// TIA Portal project "Marmita CAPIC" (V14)

(* hardware
DEVICE "S7-1200 station_1"  S7-1200 Station
   slot 0: "Rack_0"  S7-1200 Rack  Rack  V1.0
   slot 1: "Marmita CAPIC"  CPU 1214C DC/DC/DC  6ES7 214-1AG40-0XB0  V4.2
   slot 2: "DI 16/DQ 16x24VDC_1"  6ES7 223-1BL32-0XB0  V2.0
   slot 3: "DI 16/DQ 16x24VDC_2"  6ES7 223-1BL32-0XB0  V2.0
   slot 4: "AI 8xRTD_1"  SM 1231 AI8 x RTD  6ES7 231-5PF32-0XB0  V2.0
   slot 5: "AI 4x13BIT_1"  6ES7 231-4HD32-0XB0  V2.0
   slot 6: "AQ 4x14BIT_1"  6ES7 232-4HD32-0XB0  V2.0
DEVICE "CSM"  SCALANCE X-Station
   slot 0: "Bastidor SCALANCE X"  Rail
   slot 0: "Switch_MARMITA"  6GK7 277-1AA10-0AA0
DEVICE "CSM_1"  SCALANCE X-Station
   slot 0: "Bastidor SCALANCE X"  Rail
   slot 0: "Switch_REFRIGERACION"  6GK7 277-1AA10-0AA0
DEVICE "HMI MARMITA CAPIC"  Dummy PC
   slot 1: "Interfaz PROFINET"  PN-IO
*)

// ===== PLC "Marmita CAPIC"  CPU 1214C DC/DC/DC =====

VAR_GLOBAL   // PLC tag table "Tabla de variables estándar"
   "Clock_Byte" AT %MB4000 : Byte;
   "Clock_10Hz" AT %M4000.0 : Bool;
   "Clock_5Hz" AT %M4000.1 : Bool;
   "Clock_2.5Hz" AT %M4000.2 : Bool;
   "Clock_2Hz" AT %M4000.3 : Bool;
   "Clock_1.25Hz" AT %M4000.4 : Bool;
   "Clock_1Hz" AT %M4000.5 : Bool;
   "Clock_0.625Hz" AT %M4000.6 : Bool;
   "Clock_0.5Hz" AT %M4000.7 : Bool;
   "System_Byte" AT %MB4001 : Byte;
   "FirstScan" AT %M4001.0 : Bool;
   "DiagStatusUpdate" AT %M4001.1 : Bool;
   "AlwaysTRUE" AT %M4001.2 : Bool;
   "AlwaysFALSE" AT %M4001.3 : Bool;
   "Flanc_Trig_P (1Hz)" AT %M0.1 : Bool;
   "m_Zumbador" AT %M0.2 : Bool;
END_VAR

VAR_GLOBAL   // PLC tag table "Entrades Digitals"
   "Elevador abaix" AT %I8.0 : Bool;
   "Elevador adalt" AT %I8.1 : Bool;
   "Marmita volcada" AT %I8.2 : Bool;
   "Marmita desvolcada" AT %I8.3 : Bool;
   "Tapa oberta" AT %I8.4 : Bool;
   "Tapa tancada" AT %I8.5 : Bool;
   "Sensor posicio pales" AT %I8.6 : Bool;
   "Modul XPS-DMB Elevador OK" AT %I0.0 : Bool;
   "Modul XPS-DMB Tapa OK" AT %I0.1 : Bool;
   "Modul XPS-AF P.E OK" AT %I0.2 : Bool;
   "Fallo Murr" AT %I0.3 : Bool;
   "Termistor motor pales" AT %I0.4 : Bool;
   "Termistor motor volcador" AT %I0.5 : Bool;
   "Fallo Magnetotermic variador pales" AT %I0.6 : Bool;
   "Fallo Magnetotermic variador volcador" AT %I0.7 : Bool;
   "Fallo Variador pales" AT %I1.0 : Bool;
   "Fallo Variador volcador" AT %I1.1 : Bool;
   "MARXA PROCES" AT %I10.0 : Bool;
   "PARADA PROCES" AT %I10.1 : Bool;
   "PAUSA PROCES" AT %I10.2 : Bool;
   "CT100 Contador Entrada Aigua Osmotitzada" AT %I1.5 : Bool;   // 1 impuls = 1 L
   "Boto Pujar Elevador" AT %I10.3 : Bool;
   "Boto Paro Elevador" AT %I10.4 : Bool;
   "Boto Baixar Elevador" AT %I10.5 : Bool;
   "Boto volcar marmita" AT %I10.6 : Bool;
   "Boto desvolcar marmita" AT %I10.7 : Bool;
   "Boto pujar tapa" AT %I11.0 : Bool;
   "Boto baixar tapa" AT %I11.1 : Bool;
   "Boto marxa pales" AT %I11.2 : Bool;
   "Boto paro pales" AT %I11.3 : Bool;
   "Boto marxa turmix" AT %I11.4 : Bool;
   "Boto paro turmix" AT %I11.5 : Bool;
   "Fallo Termic Elevador" AT %I1.2 : Bool;
END_VAR

VAR_GLOBAL   // PLC tag table "Sortides Digitals"
   "Color Verd" AT %Q0.0 : Bool;
   "Color Taronja" AT %Q0.1 : Bool;
   "Color Vermell" AT %Q0.2 : Bool;
   "Zumbador" AT %Q0.3 : Bool;
   "Pujar Elevador" AT %Q8.0 : Bool;
   "Baixar Elevador" AT %Q8.1 : Bool;
   "Volcar Marmita" AT %Q8.2 : Bool;
   "Desvolcar Marmita" AT %Q8.3 : Bool;
   "Pujar Tapa" AT %Q8.4 : Bool;
   "Baixar Tapa" AT %Q8.5 : Bool;
   "Motor Pales" AT %Q8.6 : Bool;
   "Motor Turmix" AT %Q8.7 : Bool;
   "EV Aire Comprimit" AT %Q9.0 : Bool;
   "EV107 Purga Camisa" AT %Q9.2 : Bool;
   "EV108 Aigua Osmotitzada" AT %Q9.1 : Bool;
   "EV101 Retorn Condensats Vapor" AT %Q9.3 : Bool;
   "EV102 Entrada Aero" AT %Q9.4 : Bool;
   "EV103 Retorn Aero" AT %Q9.5 : Bool;
   "EV104 Entrada Aigua Freda" AT %Q9.6 : Bool;
   "EV105 Retorn Aigua Freda" AT %Q9.7 : Bool;
END_VAR

VAR_GLOBAL   // PLC tag table "Entrades Analogiques"
   "BT100 Sonda Tº Entrada Vapor" AT %IW162 : Int;
   "BT101 Sonda Tº Condensats Vapor" AT %IW164 : Int;
   "BT102 Sonda Tº Entrada Aero" AT %IW166 : Int;
   "BT103 Sonda Tº Retorn Aero" AT %IW168 : Int;
   "BT104 Sonda Tº Entrada Aigua Freda" AT %IW170 : Int;
   "BT105 Sonda Tº Retorn Aigua Freda" AT %IW172 : Int;
   "BP100 Presostat Entrada Vapor" AT %IW112 : Int;
   "BP101 Presostat Condensats Vapor" AT %IW114 : Int;
   "BP102 Presostat Aire" AT %IW116 : Int;
   "Sonda Temperatura Producte" AT %IW160 : Int;
END_VAR

VAR_GLOBAL   // PLC tag table "Sortides Analogiques"
   "EV100 Entrada Vapor" AT %QW176 : Int;
END_VAR

VAR_GLOBAL   // PLC tag table "PID Vapor"
   "Distrurbance" AT %MD106 : Real;
   "ManualValve" AT %MD110 : Real;
   "ErrorAck" AT %M100.0 : Bool;
   "Input_PER" AT %MW102 : Int;
   "Setpoint" AT %MD114 : Real;
   "Input" AT %MD118 : Real;
   "ManualEnable" AT %M100.1 : Bool;
   "Error" AT %M100.2 : Bool;
   "Output_PER" AT %MW104 : Int;
END_VAR

TYPE "Plantilla Variables Receptes"
   STRUCT
      Nº_Recepta : USInt;
      "Consigna Temps Inicialtizacio Hores" : USInt;
      "Consigna Temps Inicialtizacio Minuts" : USInt;
      "Consigna Temperatura" : USInt;
      "Consigna Temperatura Refredament" : USInt;
   END_STRUCT;
END_TYPE

DATA_BLOCK "DB_Recetas"   // DB2
{ S7_Optimized_Access := 'FALSE' }
VERSION : 0.1
   VAR
      "Recepta Actual" : "Plantilla Variables Receptes";
      "Recepta 1" : "Plantilla Variables Receptes";
      "Recepta 2" : "Plantilla Variables Receptes";
      "Recepta 3" : "Plantilla Variables Receptes";
      "Recepta 4" : "Plantilla Variables Receptes";
      "Recepta 5" : "Plantilla Variables Receptes";
      "Recepta 6" : "Plantilla Variables Receptes";
      "Recepta 7" : "Plantilla Variables Receptes";
      "Recepta 8" : "Plantilla Variables Receptes";
      "Recepta 9" : "Plantilla Variables Receptes";
      "Recepta 10" : "Plantilla Variables Receptes";
      "Recepta 11" : "Plantilla Variables Receptes";
      "Recepta 12" : "Plantilla Variables Receptes";
      "Recepta 13" : "Plantilla Variables Receptes";
      "Recepta 14" : "Plantilla Variables Receptes";
      "Recepta 15" : "Plantilla Variables Receptes";
      "Recepta 16" : "Plantilla Variables Receptes";
      "Recepta 17" : "Plantilla Variables Receptes";
      "Recepta 18" : "Plantilla Variables Receptes";
      "Recepta 19" : "Plantilla Variables Receptes";
      "Recepta 20" : "Plantilla Variables Receptes";
      "Recepta 21" : "Plantilla Variables Receptes";
      "Recepta 22" : "Plantilla Variables Receptes";
      "Recepta 23" : "Plantilla Variables Receptes";
      "Recepta 24" : "Plantilla Variables Receptes";
      "Recepta 25" : "Plantilla Variables Receptes";
      "Recepta 26" : "Plantilla Variables Receptes";
      "Recepta 27" : "Plantilla Variables Receptes";
      "Recepta 28" : "Plantilla Variables Receptes";
      "Recepta 29" : "Plantilla Variables Receptes";
      "Recepta 30" : "Plantilla Variables Receptes";
   END_VAR
BEGIN
END_DATA_BLOCK

DATA_BLOCK "Contador hores funcionament pales"   // DB3
{ S7_Optimized_Access := 'TRUE' }
VERSION : 0.1
// stored: InstanceOfName Contador hores de funcionament
"Contador hores de funcionament"
BEGIN
END_DATA_BLOCK

DATA_BLOCK "FB Pales_DB"   // DB4
{ S7_Optimized_Access := 'TRUE' }
VERSION : 0.1
// stored: InstanceOfName FB Pales
"FB Pales"
BEGIN
END_DATA_BLOCK

DATA_BLOCK "Control Coccio_DB"   // DB5
{ S7_Optimized_Access := 'TRUE' }
VERSION : 0.1
// stored: InstanceOfName Control Coccio
"Control Coccio"
BEGIN
END_DATA_BLOCK

DATA_BLOCK "Asignar Receptes_DB"   // DB6
{ S7_Optimized_Access := 'FALSE' }
VERSION : 0.1
// stored: InstanceOfName Asignar Receptes
"Asignar Receptes"
BEGIN
END_DATA_BLOCK

DATA_BLOCK "Intermitencia Ajustable_Zumbador_Fase_1"   // DB7
{ S7_Optimized_Access := 'TRUE' }
VERSION : 0.1
// stored: InstanceOfName Intermitencia Ajustable
"Intermitencia Ajustable"
BEGIN
END_DATA_BLOCK

DATA_BLOCK "DB_Variables_Estats"   // DB11
{ S7_Optimized_Access := 'FALSE' }
VERSION : 0.1
   VAR
      Control_Coccio : Struct
         "Estat Proces" : Bool;
         "Status Proces" : String;
      END_STRUCT;
   END_VAR
BEGIN
END_DATA_BLOCK

DATA_BLOCK "Contador aigua osmotitzada_DB"   // DB13
{ S7_Optimized_Access := 'TRUE' }
VERSION : 0.1
// stored: InstanceOfName Contador aigua osmotitzada
"Contador aigua osmotitzada"
BEGIN
END_DATA_BLOCK

DATA_BLOCK "DB_Varaibles_Pantalla"   // DB14
{ S7_Optimized_Access := 'FALSE' }
VERSION : 0.1
   VAR
      "Botons Generals" : Struct
         "Cargar Receta" : Bool;   // Carrega la recepta
      END_STRUCT;
      "Contador aigua osmotitzada" : Struct
         "Marxa Entrada Aigua" : Bool;   // Aigua osmotitzada
         "Paro Entrada Aigua" : Bool;   // Aigua osmotitzada
         "Reset Contador" : Bool;
         "Consigna Litros para Entrar" : SInt;
         "Valor contador" : SInt;
      END_STRUCT;
      "Ajustes Cocció" : Struct
         "Temps de Neteja" : SInt := 120;   // Temps de proces de neteja (segons)
      END_STRUCT;
      "Botons Manual" : Struct
         "Modo Manual" : Bool;
         "Pujar Elevador" : Bool;
         "Baixar Elevador" : Bool;
         "Volcar marmita" : Bool;
         "Desvolcar marmita" : Bool;
         "Pujar tapa" : Bool;
         "Baixar tapa" : Bool;
         "Pales ON/OFF" : Bool;
         "Tuemix ON/OFF" : Bool;
         "EV Aire" : Bool;
         "EV Aigua Freda" : Bool;
         "EV Aero" : Bool;
         "EV Purga" : Bool;
         "EV Aigua osmotitzada" : Bool;
      END_STRUCT;
   END_VAR
BEGIN
END_DATA_BLOCK

// folder: System blocks/Program resources

DATA_BLOCK "Timer_1"   // DB8
{ S7_Optimized_Access := 'TRUE' }
AUTHOR : Simatic
FAMILY : IEC
NAME : IEC_TMR
VERSION : 1.0
// stored: InstanceOfName IEC_TIMER
"IEC_TIMER"
BEGIN
END_DATA_BLOCK

DATA_BLOCK "Timer_2"   // DB9
{ S7_Optimized_Access := 'TRUE' }
AUTHOR : Simatic
FAMILY : IEC
NAME : IEC_TMR
VERSION : 1.0
// stored: InstanceOfName IEC_TIMER
"IEC_TIMER"
BEGIN
END_DATA_BLOCK

DATA_BLOCK "TM_Impuls"   // DB17
{ S7_Optimized_Access := 'TRUE' }
AUTHOR : Simatic
FAMILY : IEC
NAME : IEC_TMR
VERSION : 1.0
// stored: InstanceOfName IEC_TIMER
"IEC_TIMER"
BEGIN
END_DATA_BLOCK

// folder: (top level)

FUNCTION_BLOCK "Contador hores de funcionament"   // FB1, LAD
{ S7_Optimized_Access := 'TRUE' }
VERSION : 0.1
   VAR_INPUT
      "Entrada cicle 1 Hz" : Bool;
      "Variable de vigilancia" : Bool;
      "Valor de avis" : Time;
      "Reset Contador" : Bool;
   END_VAR
   VAR_OUTPUT
      "t Acumulat TIME" : Time;
      "t Acumulat DINT (ms)" : DInt;
      "t Manteniment TIME" : Time;
      "t Manteniment DINT (ms)" : DInt;
      "Avis de Manteniment" : Bool;
   END_VAR
   VAR
      Trig_Contador : Bool;
   END_VAR
   VAR RETAIN
      Val_Cont_Acumulat : DInt;
      Val_Cont_Manteniment : DInt;
   END_VAR
   VAR_TEMP
      temp : DInt;
   END_VAR
   VAR_TEMP   // added for the SCL form of the ladder/FBD networks
      _w1 : Bool;
      _w2 : Bool;
   END_VAR
BEGIN

REGION Network 1: Contador Acumulat
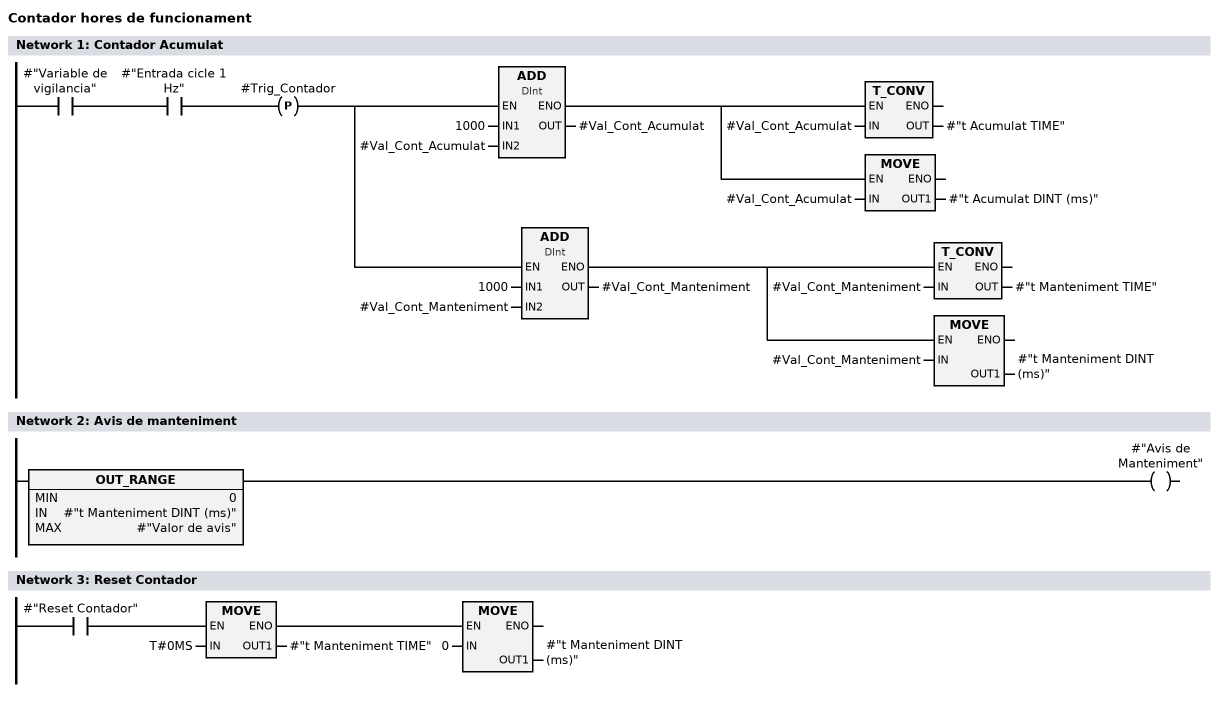
   #_w1 := #"Variable de vigilancia" AND #"Entrada cicle 1 Hz";
   #_w2 := #_w1 AND NOT #Trig_Contador;   // rising edge
   #Trig_Contador := #_w1;
   IF #_w2 THEN
       #Val_Cont_Acumulat := 1000 + #Val_Cont_Acumulat;
       #"t Acumulat TIME" := T_CONV(IN := #Val_Cont_Acumulat);
       #"t Acumulat DINT (ms)" := #Val_Cont_Acumulat;
       #Val_Cont_Manteniment := 1000 + #Val_Cont_Manteniment;
       #"t Manteniment TIME" := T_CONV(IN := #Val_Cont_Manteniment);
       #"t Manteniment DINT (ms)" := #Val_Cont_Manteniment;
   END_IF;
END_REGION

REGION Network 2: Avis de manteniment
   #"Avis de Manteniment" := (#"t Manteniment DINT (ms)" < 0) OR (#"t Manteniment DINT (ms)" > #"Valor de avis");
END_REGION

REGION Network 3: Reset Contador
   RUNG wire#powerrail
      Contact( #"Reset Contador" )
      Move(in := T#0MS, out1 => #"t Manteniment TIME")
      Move(in := 0, out1 => #"t Manteniment DINT (ms)")
   END_RUNG
   // the same network as SCL:
   IF #"Reset Contador" THEN
       #"t Manteniment TIME" := T#0MS;
       #"t Manteniment DINT (ms)" := 0;
   END_IF;
END_REGION
END_FUNCTION_BLOCK

FUNCTION_BLOCK "FB_Neteja_Camisa"   // FB2, LAD
{ S7_Optimized_Access := 'TRUE' }
VERSION : 0.1
   VAR_INPUT
      Start : Bool;
      Pausa : Bool;
      "Condicio Marxa" : Bool;
      "Clock 1 hz" : Bool;
      "Consigna Temps Neteja" : Time := T#0MS;
   END_VAR
   VAR_OUTPUT
      "EV Aire Comprimit" : Bool;
      "EV Purga" : Bool;
      Status : String;
      "Proces ON/OFF" : Bool;
      "Fin Proces" : Bool;
   END_VAR
   VAR RETAIN
      Contador_Temps_Acum : DInt;
   END_VAR
   VAR
      Trig_Start : Bool;
      Trig_1s : Bool;
      Trig_Fin : Bool;
   END_VAR
   VAR RETAIN
      En_Pausa : Bool;
      "Proces Neteja" : Bool;
   END_VAR
   VAR_TEMP
      Temp_BOOL : Bool;
      Temp_INT : Int;
      Temp_REAL : Real;
      Temp_DINT : DInt;
   END_VAR
   VAR_TEMP   // added for the SCL form of the ladder/FBD networks
      _w1 : Bool;
      _w2 : Bool;
   END_VAR
BEGIN

REGION Network 1: Inici Proces
   // Reset de Contador_Temps_Acum
   // Si condicio esta be, arranquem el proces
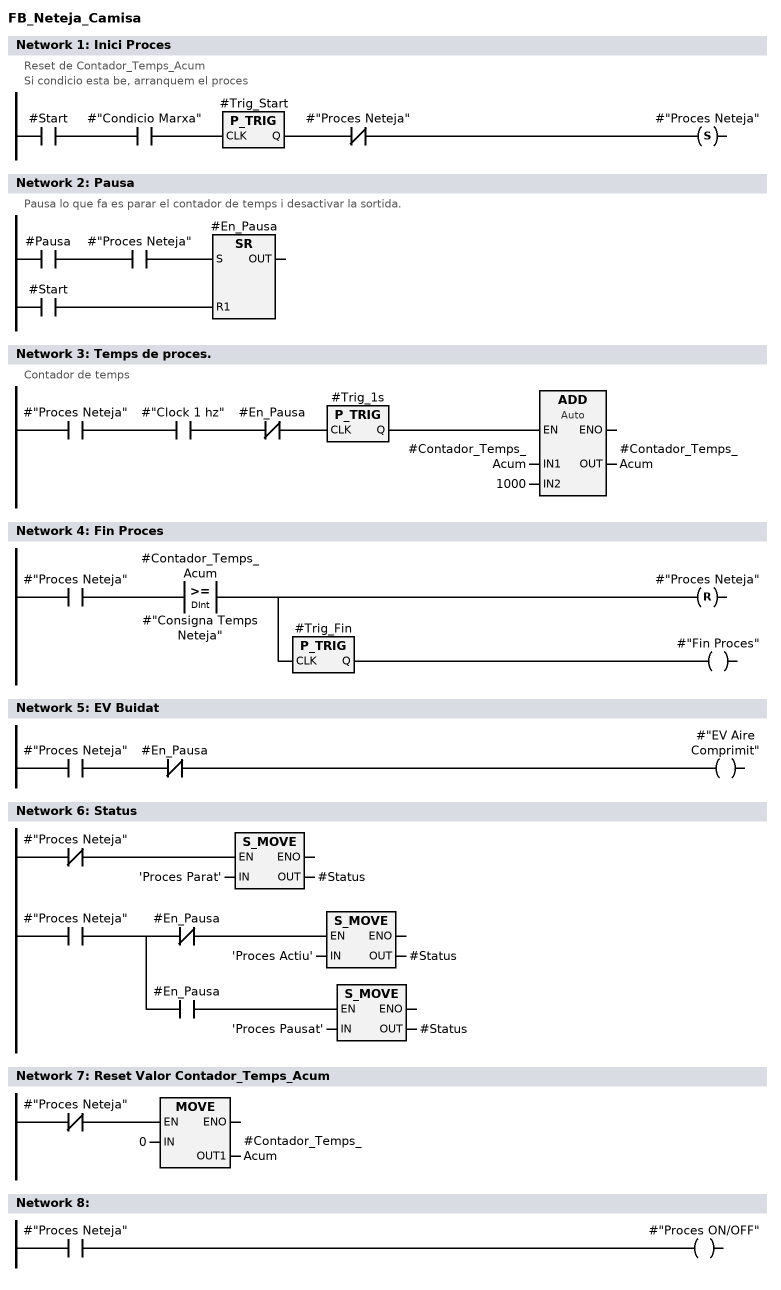
   RUNG wire#powerrail
      Contact( #Start )
      Contact( #"Condicio Marxa" )
      P_Trig( #Trig_Start )
      I_Contact( #"Proces Neteja" )
      S_Coil( #"Proces Neteja" )
   END_RUNG
   // the same network as SCL:
   #_w1 := #Start AND #"Condicio Marxa";
   #_w2 := #_w1 AND NOT #Trig_Start;   // rising edge
   #Trig_Start := #_w1;
   IF #_w2 AND NOT #"Proces Neteja" THEN #"Proces Neteja" := TRUE; END_IF;
END_REGION

REGION Network 2: Pausa
   // Pausa lo que fa es parar el contador de temps i desactivar la sortida.
   RUNG wire#powerrail
      Contact( #Pausa )
      Contact( #"Proces Neteja" )
      S_SR(operand := #En_Pausa, r1 := wire#w1)
   END_RUNG
   RUNG wire#powerrail
      Contact( #Start )
   END_RUNG wire#w1
   // the same network as SCL:
   IF #Pausa AND #"Proces Neteja" THEN
       #En_Pausa := TRUE;   // SR flip-flop
   END_IF;
   IF #Start THEN #En_Pausa := FALSE; END_IF;
END_REGION

REGION Network 3: Temps de proces.
   // Contador de temps
   RUNG wire#powerrail
      Contact( #"Proces Neteja" )
      Contact( #"Clock 1 hz" )
      I_Contact( #En_Pausa )
      P_Trig( #Trig_1s )
      Add(in1 := #Contador_Temps_Acum, in2 := 1000, out => #Contador_Temps_Acum)
   END_RUNG
   // the same network as SCL:
   #_w1 := #"Proces Neteja" AND #"Clock 1 hz" AND NOT #En_Pausa;
   #_w2 := #_w1 AND NOT #Trig_1s;   // rising edge
   #Trig_1s := #_w1;
   IF #_w2 THEN #Contador_Temps_Acum := #Contador_Temps_Acum + 1000; END_IF;
END_REGION

REGION Network 4: Fin Proces
   RUNG wire#powerrail
      Contact( #"Proces Neteja" )
      { S7_Templates := "SrcType := DInt" } GE_Contact(in1 := #Contador_Temps_Acum, in2 := #"Consigna Temps Neteja")
      wire#w1
      R_Coil( #"Proces Neteja" )
   END_RUNG
   RUNG wire#w1
      P_Trig( #Trig_Fin )
      Coil( #"Fin Proces" )
   END_RUNG
   // the same network as SCL:
   #_w1 := #"Proces Neteja" AND (#Contador_Temps_Acum >= #"Consigna Temps Neteja");
   IF #_w1 THEN #"Proces Neteja" := FALSE; END_IF;
   #_w2 := #_w1 AND NOT #Trig_Fin;   // rising edge
   #Trig_Fin := #_w1;
   #"Fin Proces" := #_w2;
END_REGION

REGION Network 5: EV Buidat
   RUNG wire#powerrail
      Contact( #"Proces Neteja" )
      I_Contact( #En_Pausa )
      Coil( #"EV Aire Comprimit" )
   END_RUNG
   // the same network as SCL:
   #"EV Aire Comprimit" := #"Proces Neteja" AND NOT #En_Pausa;
END_REGION

REGION Network 6: Status
   IF NOT #"Proces Neteja" THEN S_MOVE(in := 'Proces Parat', out => #Status); END_IF;
   IF #"Proces Neteja" AND NOT #En_Pausa THEN S_MOVE(in := 'Proces Actiu', out => #Status); END_IF;
   IF #"Proces Neteja" AND #En_Pausa THEN S_MOVE(in := 'Proces Pausat', out => #Status); END_IF;
END_REGION

REGION Network 7: Reset Valor Contador_Temps_Acum
   RUNG wire#powerrail
      I_Contact( #"Proces Neteja" )
      Move(in := 0, out1 => #Contador_Temps_Acum)
   END_RUNG
   // the same network as SCL:
   IF NOT #"Proces Neteja" THEN #Contador_Temps_Acum := 0; END_IF;
END_REGION

REGION Network 8
   RUNG wire#powerrail
      Contact( #"Proces Neteja" )
      Coil( #"Proces ON/OFF" )
   END_RUNG
   // the same network as SCL:
   #"Proces ON/OFF" := #"Proces Neteja";
END_REGION
END_FUNCTION_BLOCK

FUNCTION_BLOCK "FB Pales"   // FB4, LAD
{ S7_Optimized_Access := 'TRUE' }
VERSION : 0.1
   VAR_INPUT
      Marxa : Bool;
      Paro : Bool;
      "Condicio Marxa" : Bool;
      "Fallo Termic" : Bool;
      "Fallo Variador" : Bool;
      "Ref. Velocitat" : Int;
   END_VAR
   VAR_OUTPUT
      "Marxa Variador" : Bool;
      "OUT: Velocitat" : Int;
      "Proces ON/OFF" : Bool;
      Status : String;
   END_VAR
   VAR RETAIN
      Contador_Temps_Acum : DInt;
   END_VAR
   VAR
      Trig_Start : Bool;
      Trig_1s : Bool;
      Trig_Fin : Bool;
      "Motor Pales" : Bool;
   END_VAR
   VAR_TEMP
      Temp_Int : Int;
      Temp_Dint : DInt;
      Temp_Real : Real;
      Temp_Bool : Bool;
   END_VAR
   VAR_TEMP   // added for the SCL form of the ladder/FBD networks
      _w1 : Bool;
      _w2 : Bool;
   END_VAR
BEGIN

REGION Network 1: Inici Proces
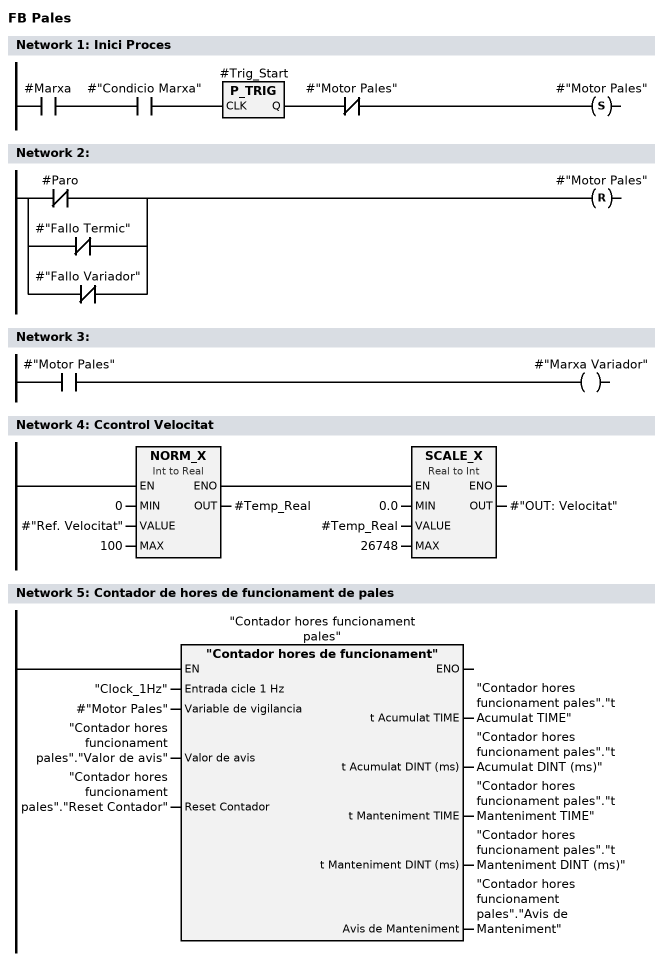
   RUNG wire#powerrail
      Contact( #Marxa )
      Contact( #"Condicio Marxa" )
      P_Trig( #Trig_Start )
      I_Contact( #"Motor Pales" )
      S_Coil( #"Motor Pales" )
   END_RUNG
   // the same network as SCL:
   #_w1 := #Marxa AND #"Condicio Marxa";
   #_w2 := #_w1 AND NOT #Trig_Start;   // rising edge
   #Trig_Start := #_w1;
   IF #_w2 AND NOT #"Motor Pales" THEN #"Motor Pales" := TRUE; END_IF;
END_REGION

REGION Network 2
   RUNG wire#powerrail
      I_Contact( #Paro )
      wire#w1
      R_Coil( #"Motor Pales" )
   END_RUNG
   RUNG wire#powerrail
      I_Contact( #"Fallo Termic" )
   END_RUNG wire#w1
   RUNG wire#powerrail
      I_Contact( #"Fallo Variador" )
   END_RUNG wire#w1
   // the same network as SCL:
   IF NOT #Paro OR NOT #"Fallo Termic" OR NOT #"Fallo Variador" THEN #"Motor Pales" := FALSE; END_IF;
END_REGION

REGION Network 3
   RUNG wire#powerrail
      Contact( #"Motor Pales" )
      Coil( #"Marxa Variador" )
   END_RUNG
   // the same network as SCL:
   #"Marxa Variador" := #"Motor Pales";
END_REGION

REGION Network 4: Ccontrol Velocitat
   RUNG wire#powerrail
      { S7_Templates := "[SrcType := Int, DestType := Real]" } Normalize(min := 0, value := #"Ref. Velocitat", max := 100, out => #Temp_Real)
      { S7_Templates := "[SrcType := Real, DestType := Int]" } Scale(min := 0.0, value := #Temp_Real, max := 26748, out => #"OUT: Velocitat")
   END_RUNG
   // the same network as SCL:
   #Temp_Real := NORM_X(MIN := 0, VALUE := #"Ref. Velocitat", MAX := 100);
   #"OUT: Velocitat" := SCALE_X(MIN := 0.0, VALUE := #Temp_Real, MAX := 26748);
END_REGION

REGION Network 5: Contador de hores de funcionament de pales
   RUNG wire#powerrail
      "Contador hores funcionament pales"("Entrada cicle 1 Hz" := "Clock_1Hz", "Variable de vigilancia" := #"Motor Pales", "Valor de avis" := "Contador hores funcionament pales"."Valor de avis", "Reset Contador" := "Contador hores funcionament pales"."Reset Contador", "t Acumulat TIME" => "Contador hores funcionament pales"."t Acumulat TIME", "t Acumulat DINT (ms)" => "Contador hores funcionament pales"."t Acumulat DINT (ms)", "t Manteniment TIME" => "Contador hores funcionament pales"."t Manteniment TIME", "t Manteniment DINT (ms)" => "Contador hores funcionament pales"."t Manteniment DINT (ms)", "Avis de Manteniment" => "Contador hores funcionament pales"."Avis de Manteniment")
   END_RUNG
   // the same network as SCL:
   "Contador hores funcionament pales"("Entrada cicle 1 Hz" := "Clock_1Hz",   // "Contador hores de funcionament"
                           "Variable de vigilancia" := #"Motor Pales",
                           "Valor de avis" := "Contador hores funcionament pales"."Valor de avis",
                           "Reset Contador" := "Contador hores funcionament pales"."Reset Contador",
                           "t Acumulat TIME" => "Contador hores funcionament pales"."t Acumulat TIME",
                           "t Acumulat DINT (ms)" => "Contador hores funcionament pales"."t Acumulat DINT (ms)",
                           "t Manteniment TIME" => "Contador hores funcionament pales"."t Manteniment TIME",
                           "t Manteniment DINT (ms)" => "Contador hores funcionament pales"."t Manteniment DINT (ms)",
                           "Avis de Manteniment" => "Contador hores funcionament pales"."Avis de Manteniment");
END_REGION
END_FUNCTION_BLOCK

FUNCTION_BLOCK "Control Coccio"   // FB8, LAD
{ S7_Optimized_Access := 'TRUE' }
VERSION : 0.1
   VAR_INPUT
      START : Bool;
      STOP : Bool;
      PAUSA : Bool;
      "Silenciar Alarma" : Bool;
      "Condicio Marxa Fase 1" : Bool;
      "Condicio Marxa Fase 2" : Bool;
      "Condicio Marxa Fase 3" : Bool;
      "Condicio Marxa Fase 4" : Bool;
      "Condicio Marxa Fase 5" : Bool;
      "Condicio Marxa Fase 6" : Bool;
      "Sonda Temperatura Producte" : USInt := 0;
      "Clock 1Hz" : Bool;
      "Receta Actual" : "Plantilla Variables Receptes";
      "Consigna Temps Neteja" : UDInt := 120;
   END_VAR
   VAR_OUTPUT
      "Estat Proces" : Bool;
      "Status Proces" : String;
   END_VAR
   VAR_IN_OUT
      Zumbador : Bool;
   END_VAR
   VAR
      M_Zumbador_Fase_1 : Bool;   // Zumbador de Avis de fin de fases i fin de procesos.
      M_Zumbador_Fase_2 : Bool;
      M_Zumbador_Fase_3 : Bool;
      M_Zumbador_Fase_4 : Bool;
      M_Zumbador_Fase_5 : Bool;
      M_Zumbador_Fase_6 : Bool;
      M_Zumbador_Fase_7 : Bool;
      M_Zumbador_Fase_8 : Bool;
      M_Zumbador_Fase_9 : Bool;
      M_Zumbador_Fase_10 : Bool;
   END_VAR
   VAR RETAIN
      M_Start : Bool;
      M_Pausa : Bool;
      "Nº Proces Actual" : USInt := 0;
      "Contador Fase 1" : UDInt;
      "Contador Fase 2" : UDInt;
      "Contador Fase 3" : UDInt;
      "Contador Fase 4" : UDInt;
      "Contador Fase 5" : UDInt;
      "Contador Fase 6" : UDInt;
      "Contador Fase 7" : UDInt;
      "Contador Fase 8" : UDInt;
      "Contador Fase 9" : UDInt;
      "Contador Fase 10" : UDInt;
      SR_Fase_1 : Bool;
      SR_Fase_2 : Bool;
      SR_Fase_3 : Bool;
      SR_Fase_4 : Bool;
      SR_Fase_5 : Bool;
      SR_Fase_6 : Bool;
      SR_Fase_7 : Bool;
      SR_Fase_8 : Bool;
      SR_Fase_9 : Bool;
      SR_Fase_10 : Bool;
   END_VAR
   VAR
      Flanc_inici_programa : Bool;
      Flanc_pausa_OFF : Bool;
      Flanc_Add_Fase_1 : Bool;
      Flanc_Add_Fase_2 : Bool;
      Flanc_Add_Fase_3 : Bool;
      Flanc_Add_Fase_4 : Bool;
      Flanc_Add_Fase_5 : Bool;
      Flanc_Add_Fase_6 : Bool;
      Flanc_Add_Fase_7 : Bool;
      Flanc_Add_Fase_8 : Bool;
      Flanc_Add_Fase_9 : Bool;
      Flanc_Add_Fase_10 : Bool;
      Buffer_Sonda_Temperatura_Producte : USInt;
      Intermitencia : Bool;
      Temp_MAX : USInt;
      "Temperatura Estable" : Bool;
   END_VAR
   VAR RETAIN
      "Conv Temps a segons" : UDInt;
   END_VAR
   VAR_TEMP
      Temp_TIME : Time;
      Temp_USINT : USInt;
   END_VAR
   VAR_TEMP   // added for the SCL form of the ladder/FBD networks
      _w1 : Bool;
      _w2 : Bool;
      _w3 : Bool;
      _w4 : Bool;
   END_VAR
BEGIN

REGION Network 1: Marxa sequencia.
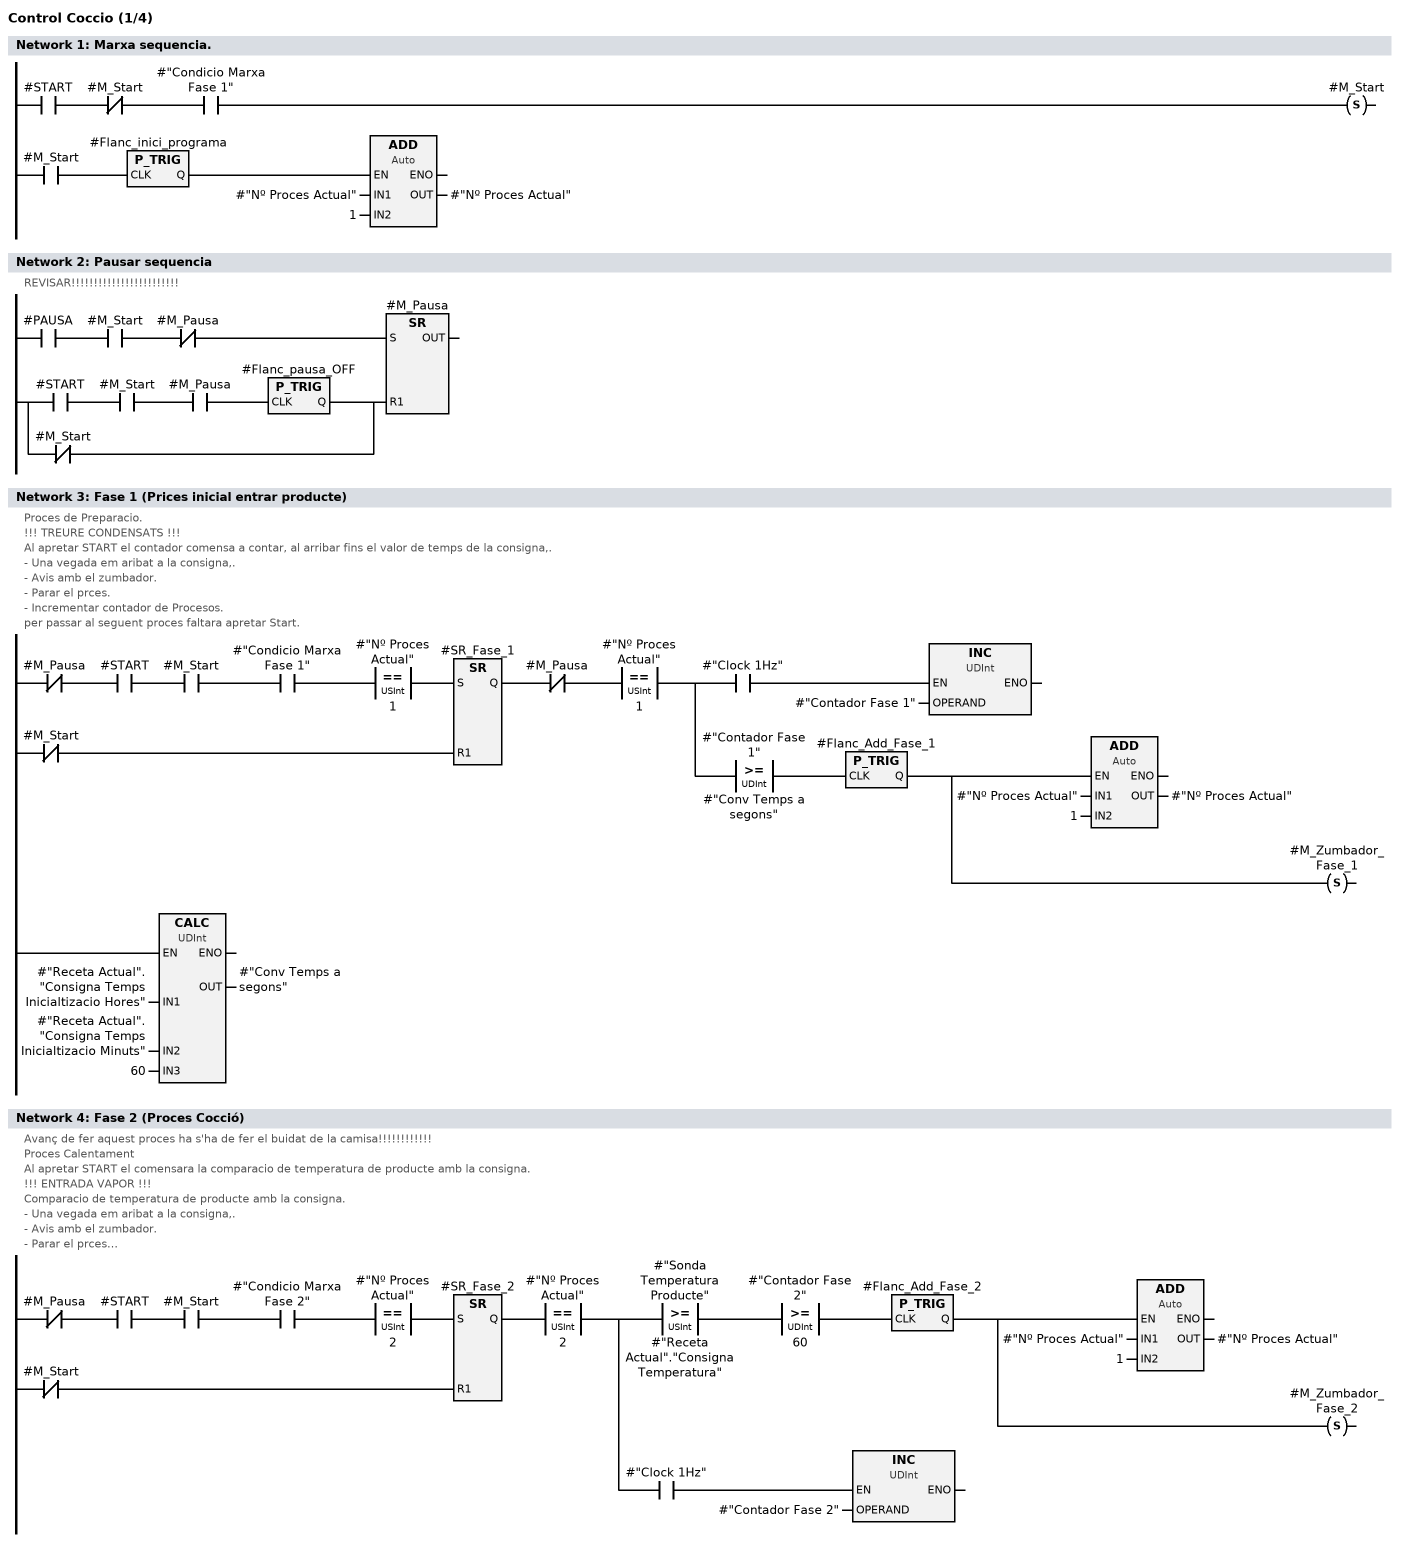
   RUNG wire#powerrail
      Contact( #START )
      I_Contact( #M_Start )
      Contact( #"Condicio Marxa Fase 1" )
      S_Coil( #M_Start )
   END_RUNG
   RUNG wire#powerrail
      Contact( #M_Start )
      P_Trig( #Flanc_inici_programa )
      Add(in1 := #"Nº Proces Actual", in2 := 1, out => #"Nº Proces Actual")
   END_RUNG
   // the same network as SCL:
   IF #START AND NOT #M_Start AND #"Condicio Marxa Fase 1" THEN #M_Start := TRUE; END_IF;
   #_w1 := #M_Start AND NOT #Flanc_inici_programa;   // rising edge
   #Flanc_inici_programa := #M_Start;
   IF #_w1 THEN #"Nº Proces Actual" := #"Nº Proces Actual" + 1; END_IF;
END_REGION

REGION Network 2: Pausar sequencia
   // REVISAR!!!!!!!!!!!!!!!!!!!!!!!!
   RUNG wire#powerrail
      Contact( #PAUSA )
      Contact( #M_Start )
      I_Contact( #M_Pausa )
      S_SR(operand := #M_Pausa, r1 := wire#w1)
   END_RUNG
   RUNG wire#powerrail
      Contact( #START )
      Contact( #M_Start )
      Contact( #M_Pausa )
      P_Trig( #Flanc_pausa_OFF )
   END_RUNG wire#w1
   RUNG wire#powerrail
      I_Contact( #M_Start )
   END_RUNG wire#w1
   // the same network as SCL:
   #_w1 := #START AND #M_Start AND #M_Pausa;
   #_w2 := #_w1 AND NOT #Flanc_pausa_OFF;   // rising edge
   #Flanc_pausa_OFF := #_w1;
   IF #PAUSA AND #M_Start AND NOT #M_Pausa THEN
       #M_Pausa := TRUE;   // SR flip-flop
   END_IF;
   IF #_w2 OR NOT #M_Start THEN #M_Pausa := FALSE; END_IF;
END_REGION

REGION Network 3: Fase 1 (Prices inicial entrar producte)
   // Proces de Preparacio.
   // 
   // !!! TREURE CONDENSATS !!!
   // 
   // Al apretar START el contador comensa a contar, al arribar fins el valor de temps de la consigna,.
   // 
   // - Una vegada em aribat a la consigna,.
   // - Avis amb el zumbador.
   // - Parar el prces.
   // - Incrementar contador de Procesos.
   // 
   // per passar al seguent proces faltara apretar Start.
   IF NOT #M_Pausa AND #START AND #M_Start AND #"Condicio Marxa Fase 1" AND (#"Nº Proces Actual" = 1) THEN
       #SR_Fase_1 := TRUE;   // SR flip-flop
   END_IF;
   IF NOT #M_Start THEN #SR_Fase_1 := FALSE; END_IF;
   #_w1 := #SR_Fase_1 AND NOT #M_Pausa AND (#"Nº Proces Actual" = 1);
   IF #_w1 AND #"Clock 1Hz" THEN #"Contador Fase 1" := #"Contador Fase 1" + 1; END_IF;
   #_w2 := #_w1 AND (#"Contador Fase 1" >= #"Conv Temps a segons");
   #_w3 := #_w2 AND NOT #Flanc_Add_Fase_1;   // rising edge
   #Flanc_Add_Fase_1 := #_w2;
   IF #_w3 THEN
       #"Nº Proces Actual" := #"Nº Proces Actual" + 1;
       #M_Zumbador_Fase_1 := TRUE;
   END_IF;
   CALC(in1 := #"Receta Actual"."Consigna Temps Inicialtizacio Hores",
        in2 := #"Receta Actual"."Consigna Temps Inicialtizacio Minuts",
        in3 := 60,
        out => #"Conv Temps a segons");
END_REGION

REGION Network 4: Fase 2 (Proces Cocció)
   // Avanç de fer aquest proces ha s'ha de fer el buidat de la camisa!!!!!!!!!!!!
   // 
   // Proces Calentament
   // 
   // Al apretar START el comensara la comparacio de temperatura de producte amb la consigna.
   // 
   // !!! ENTRADA VAPOR !!!
   // 
   // Comparacio de temperatura de producte amb la consigna.
   // 
   // - Una vegada em aribat a la consigna,.
   // - Avis amb el zumbador.
   // - Parar el prces.
   // - Incrementar contador de Procesos.
   RUNG wire#powerrail
      I_Contact( #M_Pausa )
      Contact( #START )
      Contact( #M_Start )
      Contact( #"Condicio Marxa Fase 2" )
      { S7_Templates := "SrcType := USInt" } EQ_Contact(in1 := #"Nº Proces Actual", in2 := 2)
      S_SR(operand := #SR_Fase_2, r1 := wire#w1)
      { S7_Templates := "SrcType := USInt" } EQ_Contact(in1 := #"Nº Proces Actual", in2 := 2)
      wire#w2
      { S7_Templates := "SrcType := USInt" } GE_Contact(in1 := #"Sonda Temperatura Producte", in2 := #"Receta Actual"."Consigna Temperatura")
      { S7_Templates := "SrcType := UDInt" } GE_Contact(in1 := #"Contador Fase 2", in2 := 60)
      P_Trig( #Flanc_Add_Fase_2 )
      wire#w3
      Add(in1 := #"Nº Proces Actual", in2 := 1, out => #"Nº Proces Actual")
   END_RUNG
   RUNG wire#powerrail
      I_Contact( #M_Start )
   END_RUNG wire#w1
   RUNG wire#w3
      S_Coil( #M_Zumbador_Fase_2 )
   END_RUNG
   RUNG wire#w2
      Contact( #"Clock 1Hz" )
      { S7_Templates := "DestType := UDInt" } Inc( #"Contador Fase 2" )
   END_RUNG
   // the same network as SCL:
   IF NOT #M_Pausa AND #START AND #M_Start AND #"Condicio Marxa Fase 2" AND (#"Nº Proces Actual" = 2) THEN
       #SR_Fase_2 := TRUE;   // SR flip-flop
   END_IF;
   IF NOT #M_Start THEN #SR_Fase_2 := FALSE; END_IF;
   #_w1 := #SR_Fase_2 AND (#"Nº Proces Actual" = 2);
   #_w2 := #_w1 AND (#"Sonda Temperatura Producte" >= #"Receta Actual"."Consigna Temperatura") AND (#"Contador Fase 2" >= 60);
   #_w3 := #_w2 AND NOT #Flanc_Add_Fase_2;   // rising edge
   #Flanc_Add_Fase_2 := #_w2;
   IF #_w3 THEN
       #"Nº Proces Actual" := #"Nº Proces Actual" + 1;
       #M_Zumbador_Fase_2 := TRUE;
   END_IF;
   IF #_w1 AND #"Clock 1Hz" THEN #"Contador Fase 2" := #"Contador Fase 2" + 1; END_IF;
END_REGION

REGION Network 5: Fase 3 (Neteja)
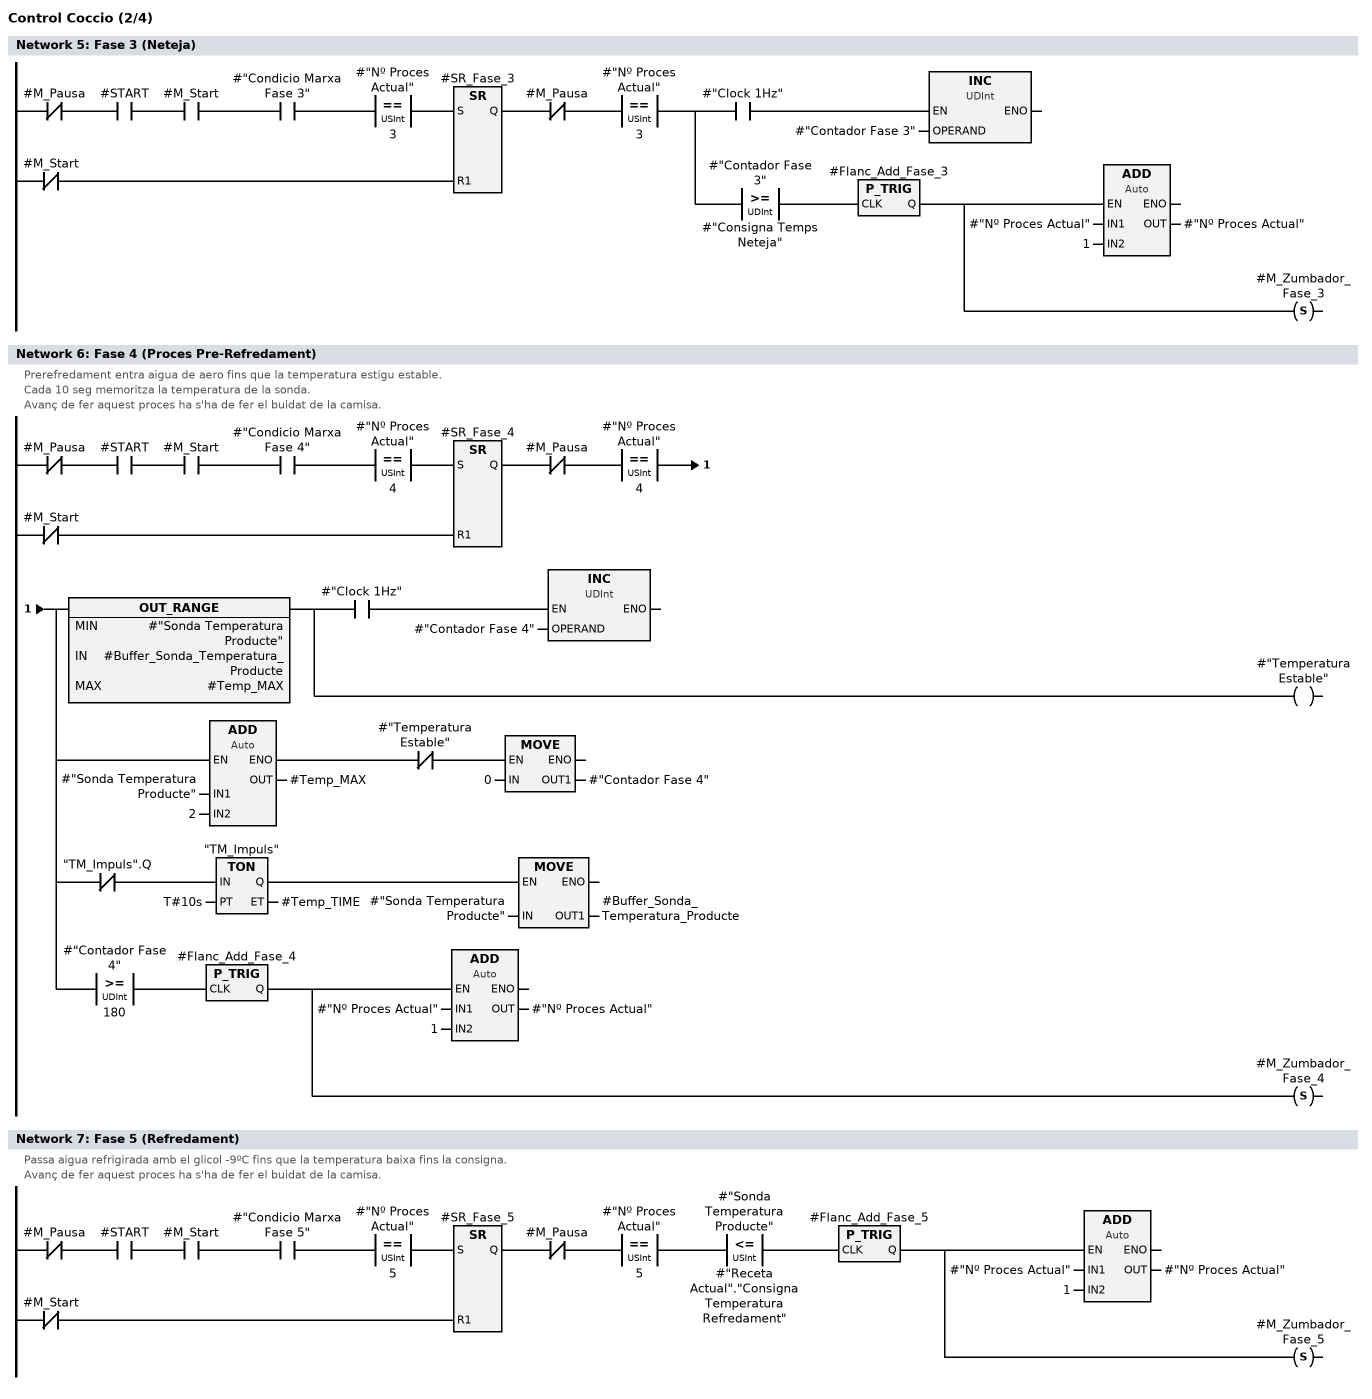
   RUNG wire#powerrail
      I_Contact( #M_Pausa )
      Contact( #START )
      Contact( #M_Start )
      Contact( #"Condicio Marxa Fase 3" )
      { S7_Templates := "SrcType := USInt" } EQ_Contact(in1 := #"Nº Proces Actual", in2 := 3)
      S_SR(operand := #SR_Fase_3, r1 := wire#w1)
      I_Contact( #M_Pausa )
      { S7_Templates := "SrcType := USInt" } EQ_Contact(in1 := #"Nº Proces Actual", in2 := 3)
      wire#w2
      Contact( #"Clock 1Hz" )
      { S7_Templates := "DestType := UDInt" } Inc( #"Contador Fase 3" )
   END_RUNG
   RUNG wire#powerrail
      I_Contact( #M_Start )
   END_RUNG wire#w1
   RUNG wire#w2
      { S7_Templates := "SrcType := UDInt" } GE_Contact(in1 := #"Contador Fase 3", in2 := #"Consigna Temps Neteja")
      P_Trig( #Flanc_Add_Fase_3 )
      wire#w3
      Add(in1 := #"Nº Proces Actual", in2 := 1, out => #"Nº Proces Actual")
   END_RUNG
   RUNG wire#w3
      S_Coil( #M_Zumbador_Fase_3 )
   END_RUNG
   // the same network as SCL:
   IF NOT #M_Pausa AND #START AND #M_Start AND #"Condicio Marxa Fase 3" AND (#"Nº Proces Actual" = 3) THEN
       #SR_Fase_3 := TRUE;   // SR flip-flop
   END_IF;
   IF NOT #M_Start THEN #SR_Fase_3 := FALSE; END_IF;
   #_w1 := #SR_Fase_3 AND NOT #M_Pausa AND (#"Nº Proces Actual" = 3);
   IF #_w1 AND #"Clock 1Hz" THEN #"Contador Fase 3" := #"Contador Fase 3" + 1; END_IF;
   #_w2 := #_w1 AND (#"Contador Fase 3" >= #"Consigna Temps Neteja");
   #_w3 := #_w2 AND NOT #Flanc_Add_Fase_3;   // rising edge
   #Flanc_Add_Fase_3 := #_w2;
   IF #_w3 THEN
       #"Nº Proces Actual" := #"Nº Proces Actual" + 1;
       #M_Zumbador_Fase_3 := TRUE;
   END_IF;
END_REGION

REGION Network 6: Fase 4 (Proces Pre-Refredament)
   // Prerefredament entra aigua de aero fins que la temperatura estigu estable.
   // 
   // Cada 10 seg memoritza la temperatura de la sonda.
   // 
   // Avanç de fer aquest proces ha s'ha de fer el buidat de la camisa.
   IF NOT #M_Pausa AND #START AND #M_Start AND #"Condicio Marxa Fase 4" AND (#"Nº Proces Actual" = 4) THEN
       #SR_Fase_4 := TRUE;   // SR flip-flop
   END_IF;
   IF NOT #M_Start THEN #SR_Fase_4 := FALSE; END_IF;
   #_w1 := #SR_Fase_4 AND NOT #M_Pausa AND (#"Nº Proces Actual" = 4);
   #_w2 := #_w1 AND ((#Buffer_Sonda_Temperatura_Producte < #"Sonda Temperatura Producte") OR (#Buffer_Sonda_Temperatura_Producte > #Temp_MAX));
   IF #_w2 AND #"Clock 1Hz" THEN #"Contador Fase 4" := #"Contador Fase 4" + 1; END_IF;
   #"Temperatura Estable" := #_w2;
   IF #_w1 THEN #Temp_MAX := #"Sonda Temperatura Producte" + 2; END_IF;
   IF #_w1 AND NOT #"Temperatura Estable" THEN #"Contador Fase 4" := 0; END_IF;
   "TM_Impuls".TON(IN := #_w1 AND NOT "TM_Impuls".Q, PT := T#10s, ET => #Temp_TIME);
   IF "TM_Impuls".Q THEN #Buffer_Sonda_Temperatura_Producte := #"Sonda Temperatura Producte"; END_IF;
   #_w3 := #_w1 AND (#"Contador Fase 4" >= 180);
   #_w4 := #_w3 AND NOT #Flanc_Add_Fase_4;   // rising edge
   #Flanc_Add_Fase_4 := #_w3;
   IF #_w4 THEN
       #"Nº Proces Actual" := #"Nº Proces Actual" + 1;
       #M_Zumbador_Fase_4 := TRUE;
   END_IF;
END_REGION

REGION Network 7: Fase 5 (Refredament)
   // Passa aigua refrigirada amb el glicol -9ºC fins que la temperatura baixa fins la consigna.
   // 
   // Avanç de fer aquest proces ha s'ha de fer el buidat de la camisa.
   RUNG wire#powerrail
      I_Contact( #M_Pausa )
      Contact( #START )
      Contact( #M_Start )
      Contact( #"Condicio Marxa Fase 5" )
      { S7_Templates := "SrcType := USInt" } EQ_Contact(in1 := #"Nº Proces Actual", in2 := 5)
      S_SR(operand := #SR_Fase_5, r1 := wire#w1)
      I_Contact( #M_Pausa )
      { S7_Templates := "SrcType := USInt" } EQ_Contact(in1 := #"Nº Proces Actual", in2 := 5)
      { S7_Templates := "SrcType := USInt" } LE_Contact(in1 := #"Sonda Temperatura Producte", in2 := #"Receta Actual"."Consigna Temperatura Refredament")
      P_Trig( #Flanc_Add_Fase_5 )
      wire#w2
      Add(in1 := #"Nº Proces Actual", in2 := 1, out => #"Nº Proces Actual")
   END_RUNG
   RUNG wire#powerrail
      I_Contact( #M_Start )
   END_RUNG wire#w1
   RUNG wire#w2
      S_Coil( #M_Zumbador_Fase_5 )
   END_RUNG
   // the same network as SCL:
   IF NOT #M_Pausa AND #START AND #M_Start AND #"Condicio Marxa Fase 5" AND (#"Nº Proces Actual" = 5) THEN
       #SR_Fase_5 := TRUE;   // SR flip-flop
   END_IF;
   IF NOT #M_Start THEN #SR_Fase_5 := FALSE; END_IF;
   #_w1 := #SR_Fase_5 AND NOT #M_Pausa AND (#"Nº Proces Actual" = 5) AND (#"Sonda Temperatura Producte" <= #"Receta Actual"."Consigna Temperatura Refredament");
   #_w2 := #_w1 AND NOT #Flanc_Add_Fase_5;   // rising edge
   #Flanc_Add_Fase_5 := #_w1;
   IF #_w2 THEN
       #"Nº Proces Actual" := #"Nº Proces Actual" + 1;
       #M_Zumbador_Fase_5 := TRUE;
   END_IF;
END_REGION

REGION Network 8: Fase 6 (Neteja)
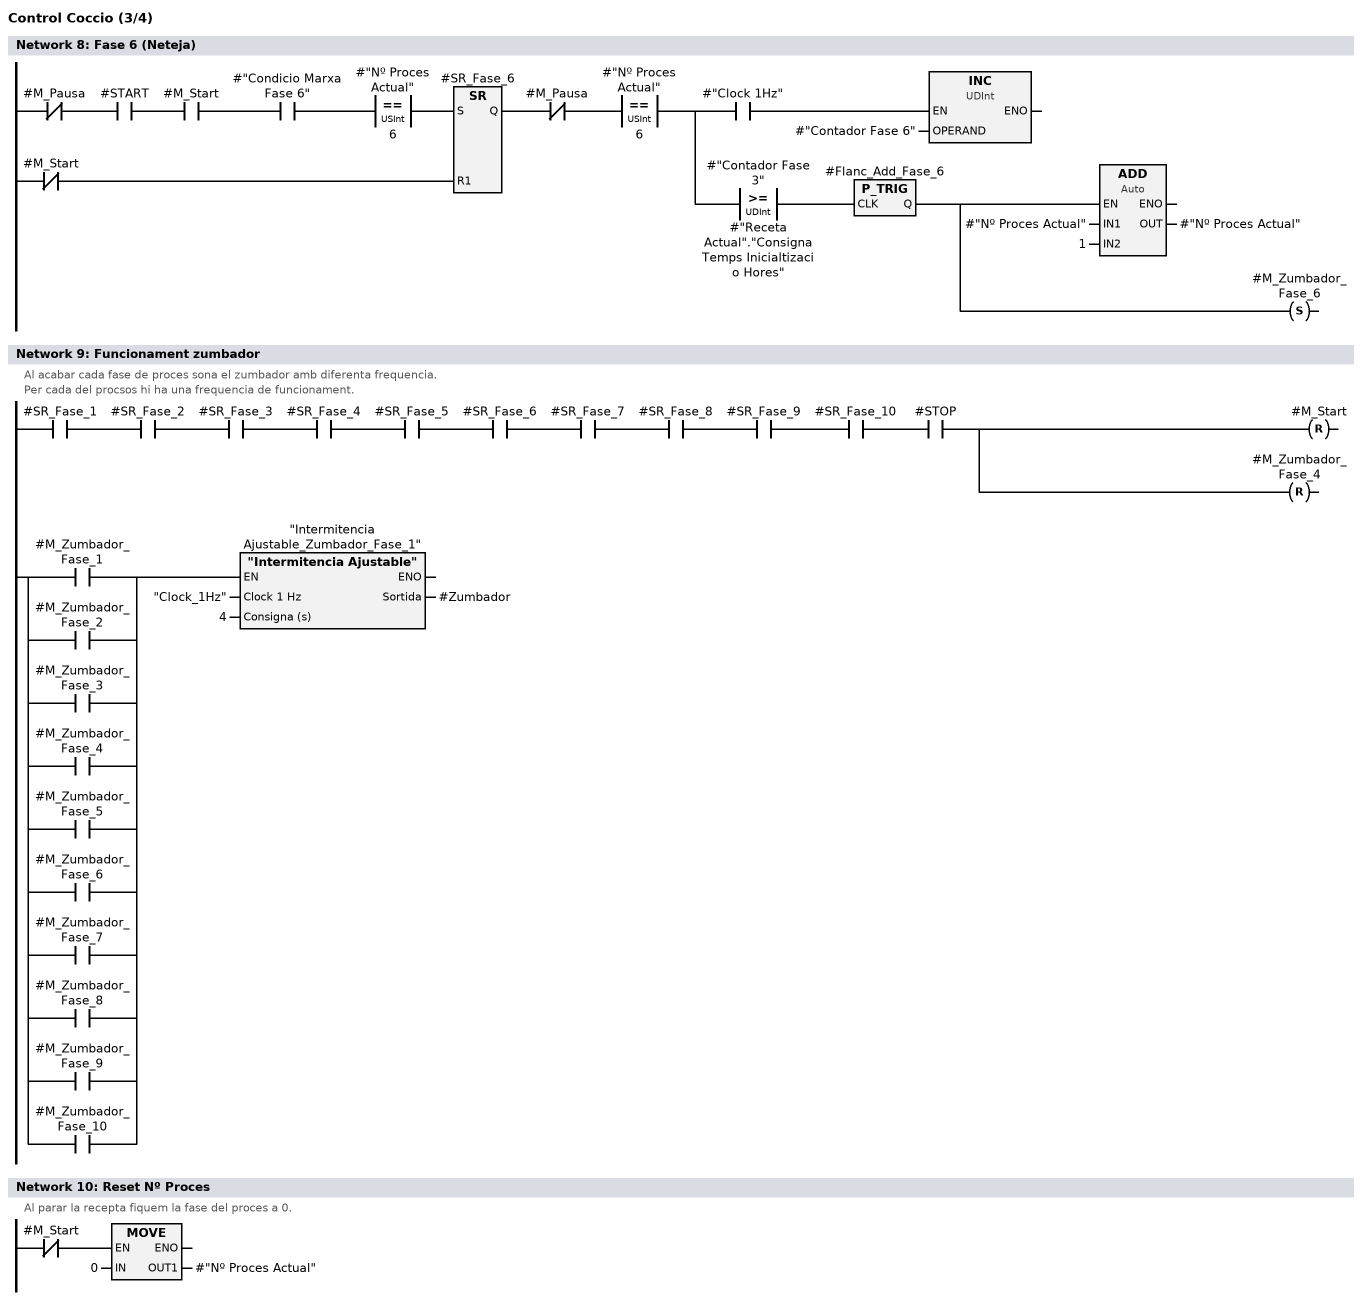
   RUNG wire#powerrail
      I_Contact( #M_Pausa )
      Contact( #START )
      Contact( #M_Start )
      Contact( #"Condicio Marxa Fase 6" )
      { S7_Templates := "SrcType := USInt" } EQ_Contact(in1 := #"Nº Proces Actual", in2 := 6)
      S_SR(operand := #SR_Fase_6, r1 := wire#w1)
      I_Contact( #M_Pausa )
      { S7_Templates := "SrcType := USInt" } EQ_Contact(in1 := #"Nº Proces Actual", in2 := 6)
      wire#w2
      Contact( #"Clock 1Hz" )
      { S7_Templates := "DestType := UDInt" } Inc( #"Contador Fase 6" )
   END_RUNG
   RUNG wire#powerrail
      I_Contact( #M_Start )
   END_RUNG wire#w1
   RUNG wire#w2
      { S7_Templates := "SrcType := UDInt" } GE_Contact(in1 := #"Contador Fase 3", in2 := #"Receta Actual"."Consigna Temps Inicialtizacio Hores")
      P_Trig( #Flanc_Add_Fase_6 )
      wire#w3
      Add(in1 := #"Nº Proces Actual", in2 := 1, out => #"Nº Proces Actual")
   END_RUNG
   RUNG wire#w3
      S_Coil( #M_Zumbador_Fase_6 )
   END_RUNG
   // the same network as SCL:
   IF NOT #M_Pausa AND #START AND #M_Start AND #"Condicio Marxa Fase 6" AND (#"Nº Proces Actual" = 6) THEN
       #SR_Fase_6 := TRUE;   // SR flip-flop
   END_IF;
   IF NOT #M_Start THEN #SR_Fase_6 := FALSE; END_IF;
   #_w1 := #SR_Fase_6 AND NOT #M_Pausa AND (#"Nº Proces Actual" = 6);
   IF #_w1 AND #"Clock 1Hz" THEN #"Contador Fase 6" := #"Contador Fase 6" + 1; END_IF;
   #_w2 := #_w1 AND (#"Contador Fase 3" >= #"Receta Actual"."Consigna Temps Inicialtizacio Hores");
   #_w3 := #_w2 AND NOT #Flanc_Add_Fase_6;   // rising edge
   #Flanc_Add_Fase_6 := #_w2;
   IF #_w3 THEN
       #"Nº Proces Actual" := #"Nº Proces Actual" + 1;
       #M_Zumbador_Fase_6 := TRUE;
   END_IF;
END_REGION

REGION Network 9: Funcionament zumbador
   // Al acabar cada fase de proces sona el zumbador amb diferenta frequencia.
   // Per cada del procsos hi ha una frequencia de funcionament.
   RUNG wire#powerrail
      Contact( #SR_Fase_1 )
      Contact( #SR_Fase_2 )
      Contact( #SR_Fase_3 )
      Contact( #SR_Fase_4 )
      Contact( #SR_Fase_5 )
      Contact( #SR_Fase_6 )
      Contact( #SR_Fase_7 )
      Contact( #SR_Fase_8 )
      Contact( #SR_Fase_9 )
      Contact( #SR_Fase_10 )
      Contact( #STOP )
      wire#w1
      R_Coil( #M_Start )
   END_RUNG
   RUNG wire#w1
      R_Coil( #M_Zumbador_Fase_4 )
   END_RUNG
   RUNG wire#powerrail
      Contact( #M_Zumbador_Fase_1 )
      wire#w2
      "Intermitencia Ajustable_Zumbador_Fase_1"("Clock 1 Hz" := "Clock_1Hz", "Consigna (s)" := 4, Sortida => #Zumbador)
   END_RUNG
   RUNG wire#powerrail
      Contact( #M_Zumbador_Fase_2 )
   END_RUNG wire#w2
   RUNG wire#powerrail
      Contact( #M_Zumbador_Fase_3 )
   END_RUNG wire#w2
   RUNG wire#powerrail
      Contact( #M_Zumbador_Fase_4 )
   END_RUNG wire#w2
   RUNG wire#powerrail
      Contact( #M_Zumbador_Fase_5 )
   END_RUNG wire#w2
   RUNG wire#powerrail
      Contact( #M_Zumbador_Fase_6 )
   END_RUNG wire#w2
   RUNG wire#powerrail
      Contact( #M_Zumbador_Fase_7 )
   END_RUNG wire#w2
   RUNG wire#powerrail
      Contact( #M_Zumbador_Fase_8 )
   END_RUNG wire#w2
   RUNG wire#powerrail
      Contact( #M_Zumbador_Fase_9 )
   END_RUNG wire#w2
   RUNG wire#powerrail
      Contact( #M_Zumbador_Fase_10 )
   END_RUNG wire#w2
   // the same network as SCL:
   IF #SR_Fase_1 AND #SR_Fase_2 AND #SR_Fase_3 AND #SR_Fase_4 AND #SR_Fase_5 AND #SR_Fase_6 AND #SR_Fase_7 AND #SR_Fase_8 AND #SR_Fase_9 AND #SR_Fase_10 AND #STOP THEN
       #M_Start := FALSE;
       #M_Zumbador_Fase_4 := FALSE;
   END_IF;
   IF #M_Zumbador_Fase_1 OR #M_Zumbador_Fase_2 OR #M_Zumbador_Fase_3 OR #M_Zumbador_Fase_4 OR #M_Zumbador_Fase_5 OR #M_Zumbador_Fase_6 OR #M_Zumbador_Fase_7 OR #M_Zumbador_Fase_8 OR #M_Zumbador_Fase_9 OR #M_Zumbador_Fase_10 THEN
       "Intermitencia Ajustable_Zumbador_Fase_1"("Clock 1 Hz" := "Clock_1Hz",   // "Intermitencia Ajustable"
                               "Consigna (s)" := 4,
                               Sortida => #Zumbador);
   END_IF;
END_REGION

REGION Network 10: Reset Nº Proces
   // Al parar la recepta fiquem la fase del proces a 0.
   RUNG wire#powerrail
      I_Contact( #M_Start )
      Move(in := 0, out1 => #"Nº Proces Actual")
   END_RUNG
   // the same network as SCL:
   IF NOT #M_Start THEN #"Nº Proces Actual" := 0; END_IF;
END_REGION

REGION Network 11: Limitacio de Nº de procesos.
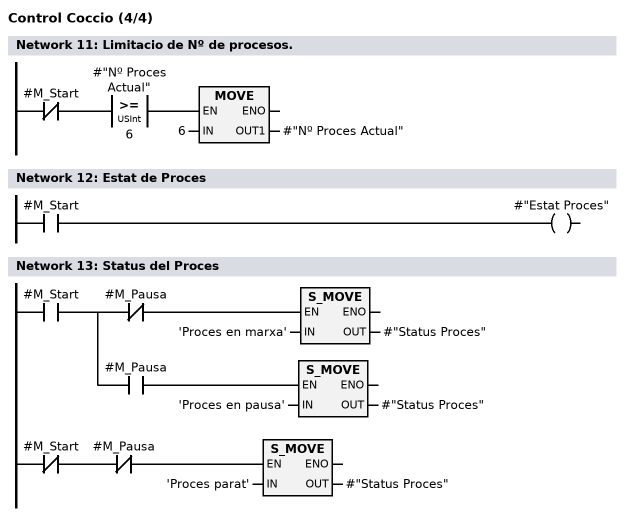
   RUNG wire#powerrail
      I_Contact( #M_Start )
      { S7_Templates := "SrcType := USInt" } GE_Contact(in1 := #"Nº Proces Actual", in2 := 6)
      Move(in := 6, out1 => #"Nº Proces Actual")
   END_RUNG
   // the same network as SCL:
   IF NOT #M_Start AND (#"Nº Proces Actual" >= 6) THEN #"Nº Proces Actual" := 6; END_IF;
END_REGION

REGION Network 12: Estat de Proces
   RUNG wire#powerrail
      Contact( #M_Start )
      Coil( #"Estat Proces" )
   END_RUNG
   // the same network as SCL:
   #"Estat Proces" := #M_Start;
END_REGION

REGION Network 13: Status del Proces
   IF #M_Start AND NOT #M_Pausa THEN S_MOVE(in := 'Proces en marxa', out => #"Status Proces"); END_IF;
   IF #M_Start AND #M_Pausa THEN S_MOVE(in := 'Proces en pausa', out => #"Status Proces"); END_IF;
   IF NOT #M_Start AND NOT #M_Pausa THEN S_MOVE(in := 'Proces parat', out => #"Status Proces"); END_IF;
END_REGION
END_FUNCTION_BLOCK

FUNCTION_BLOCK "Asignar Receptes"   // FB9, LAD
{ S7_Optimized_Access := 'FALSE' }
VERSION : 0.1
   VAR_INPUT
      "Cargar Receta" : Bool;
      "Receta a cargar" : USInt;
   END_VAR
   VAR_OUTPUT
      "Receta Actual" : USInt;
      "Nº Receta a cargar" : USInt;
      Status : String;
   END_VAR
   VAR_IN_OUT
      "Receta Acrual" : "Plantilla Variables Receptes";
   END_VAR
BEGIN

REGION Network 1 (SCL)
   // Si Cargar Receta = true , asignem de la plantilla seleccionada els valors a la "Receta Acrual"
   #"Nº Receta a cargar" := #"Receta a cargar";

   IF #"Cargar Receta" THEN
       #"Receta Actual":= #"Receta a cargar";
       #"Nº Receta a cargar" := #"Receta a cargar";
       CASE #"Receta a cargar" OF
           0:
               #Status := 'Receta no esta asignada';
               #"Receta Actual" := 0;
           1:
               #"Receta Acrual" := "DB_Recetas"."Recepta 1";
               #Status := 'Recepta 1';
           2:
               #"Receta Acrual" := "DB_Recetas"."Recepta 2";
               #Status := 'Recepta 2';
           3:
               #"Receta Acrual" := "DB_Recetas"."Recepta 3";
               #Status := 'Recepta 3';
           4:
               #"Receta Acrual" := "DB_Recetas"."Recepta 4";
               #Status := 'Recepta 4';
           5:
               #"Receta Acrual" := "DB_Recetas"."Recepta 5";
               #Status := 'Recepta 5';
           6:
               #"Receta Acrual" := "DB_Recetas"."Recepta 6";
               #Status := 'Recepta 6';
           7:
               #"Receta Acrual" := "DB_Recetas"."Recepta 7";
               #Status := 'Recepta 7';
           8:
               #"Receta Acrual" := "DB_Recetas"."Recepta 8";
               #Status := 'Recepta 8';
           9:
               #"Receta Acrual" := "DB_Recetas"."Recepta 9";
               #Status := 'Recepta 9';
           10:
               #"Receta Acrual" := "DB_Recetas"."Recepta 10";
               #Status := 'Recepta 10';
           11:
               #"Receta Acrual" := "DB_Recetas"."Recepta 11";
               #Status := 'Recepta 11';
           12:
               #"Receta Acrual" := "DB_Recetas"."Recepta 12";
               #Status := 'Recepta 12';
           13:
               #"Receta Acrual" := "DB_Recetas"."Recepta 13";
               #Status := 'Recepta 13';
           14:
               #"Receta Acrual" := "DB_Recetas"."Recepta 14";
               #Status := 'Recepta 14';
           15:
               #"Receta Acrual" := "DB_Recetas"."Recepta 15";
               #Status := 'Recepta 15';
           16:
               #"Receta Acrual" := "DB_Recetas"."Recepta 16";
               #Status := 'Recepta 16';
           17:
               #"Receta Acrual" := "DB_Recetas"."Recepta 17";
               #Status := 'Recepta 17';
           18:
               #"Receta Acrual" := "DB_Recetas"."Recepta 18";
               #Status := 'Recepta 18';
           19:
               #"Receta Acrual" := "DB_Recetas"."Recepta 19";
               #Status := 'Recepta 19';
           20:
               #"Receta Acrual" := "DB_Recetas"."Recepta 20";
               #Status := 'Recepta 20';
           21:
               #"Receta Acrual" := "DB_Recetas"."Recepta 21";
               #Status := 'Recepta 21';
           22:
               #"Receta Acrual" := "DB_Recetas"."Recepta 22";
               #Status := 'Recepta 22';
           23:
               #"Receta Acrual" := "DB_Recetas"."Recepta 23";
               #Status := 'Recepta 23';
           24:
               #"Receta Acrual" := "DB_Recetas"."Recepta 24";
               #Status := 'Recepta 24';
           25:
               #"Receta Acrual" := "DB_Recetas"."Recepta 25";
               #Status := 'Recepta 25';
           26:
               #"Receta Acrual" := "DB_Recetas"."Recepta 26";
               #Status := 'Recepta 26';
           27:
               #"Receta Acrual" := "DB_Recetas"."Recepta 27";
               #Status := 'Recepta 27';
           28:
               #"Receta Acrual" := "DB_Recetas"."Recepta 28";
               #Status := 'Recepta 28';
           29:
               #"Receta Acrual" := "DB_Recetas"."Recepta 29";
               #Status := 'Recepta 29';
           30:
               #"Receta Acrual" := "DB_Recetas"."Recepta 30";
               #Status := 'Recepta 30';

       END_CASE;
       ;
   END_IF;
END_REGION
END_FUNCTION_BLOCK

FUNCTION_BLOCK "Intermitencia Ajustable"   // FB10, LAD
{ S7_Optimized_Access := 'TRUE' }
VERSION : 0.1
   VAR_INPUT
      "Clock 1 Hz" : Bool;
      "Consigna (s)" : SInt;
   END_VAR
   VAR_OUTPUT
      Sortida : Bool;
   END_VAR
   VAR
      Flanc_inici_programa : Bool;
      contador : SInt;
   END_VAR
   VAR_TEMP
      Temp_SINT : SInt;
   END_VAR
   VAR_TEMP   // added for the SCL form of the ladder/FBD networks
      _w1 : Bool;
   END_VAR
BEGIN

REGION Network 1
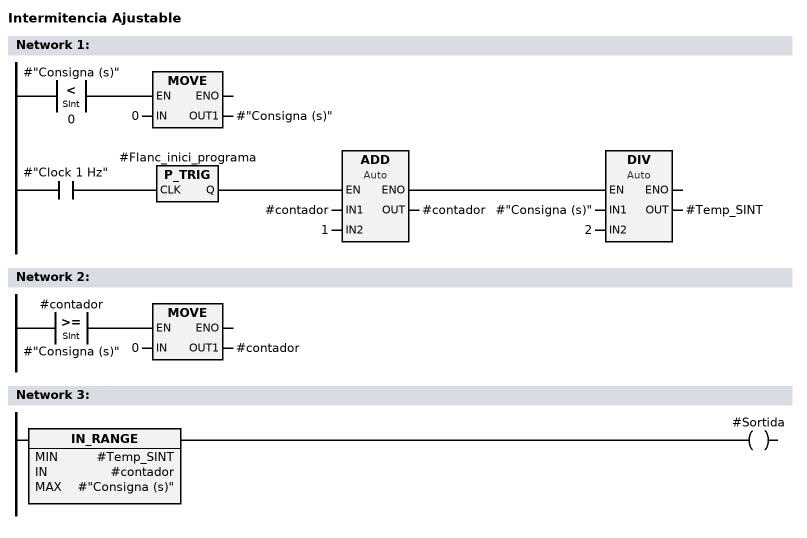
   RUNG wire#powerrail
      { S7_Templates := "SrcType := SInt" } LT_Contact(in1 := #"Consigna (s)", in2 := 0)
      Move(in := 0, out1 => #"Consigna (s)")
   END_RUNG
   RUNG wire#powerrail
      Contact( #"Clock 1 Hz" )
      P_Trig( #Flanc_inici_programa )
      Add(in1 := #contador, in2 := 1, out => #contador)
      Div(in1 := #"Consigna (s)", in2 := 2, out => #Temp_SINT)
   END_RUNG
   // the same network as SCL:
   IF #"Consigna (s)" < 0 THEN #"Consigna (s)" := 0; END_IF;
   #_w1 := #"Clock 1 Hz" AND NOT #Flanc_inici_programa;   // rising edge
   #Flanc_inici_programa := #"Clock 1 Hz";
   IF #_w1 THEN
       #contador := #contador + 1;
       #Temp_SINT := #"Consigna (s)" / 2;
   END_IF;
END_REGION

REGION Network 2
   RUNG wire#powerrail
      { S7_Templates := "SrcType := SInt" } GE_Contact(in1 := #contador, in2 := #"Consigna (s)")
      Move(in := 0, out1 => #contador)
   END_RUNG
   // the same network as SCL:
   IF #contador >= #"Consigna (s)" THEN #contador := 0; END_IF;
END_REGION

REGION Network 3
   RUNG wire#powerrail
      { S7_Templates := "SrcType := SInt" } InRange(min := #Temp_SINT, in := #contador, max := #"Consigna (s)")
      Coil( #Sortida )
   END_RUNG
   // the same network as SCL:
   #Sortida := (#Temp_SINT <= #contador) AND (#contador <= #"Consigna (s)");
END_REGION
END_FUNCTION_BLOCK

FUNCTION_BLOCK "Contador aigua osmotitzada"   // FB12, LAD
{ S7_Optimized_Access := 'TRUE' }
VERSION : 0.1
   VAR_INPUT
      Condicions : Bool;
      "Entrada impulsos" : Bool;
      Start : Bool;
      Stop : Bool;
      "Reset Contador" : Bool;
   END_VAR
   VAR_OUTPUT
      "EV Entrar Aigua" : Bool;
      "Valor Contador" : SInt;
   END_VAR
   VAR_IN_OUT
      "Consigna Litros Per Entrar" : SInt;
   END_VAR
   VAR RETAIN
      Contador : SInt;
   END_VAR
   VAR
      M_Flanc_Clock_1z : SInt;
      M_Flank_Contador : Bool;
      En_Marxa : Bool;
   END_VAR
   VAR_TEMP   // added for the SCL form of the ladder/FBD networks
      _w1 : Bool;
      _w2 : Bool;
   END_VAR
BEGIN

REGION Network 1: Marxa
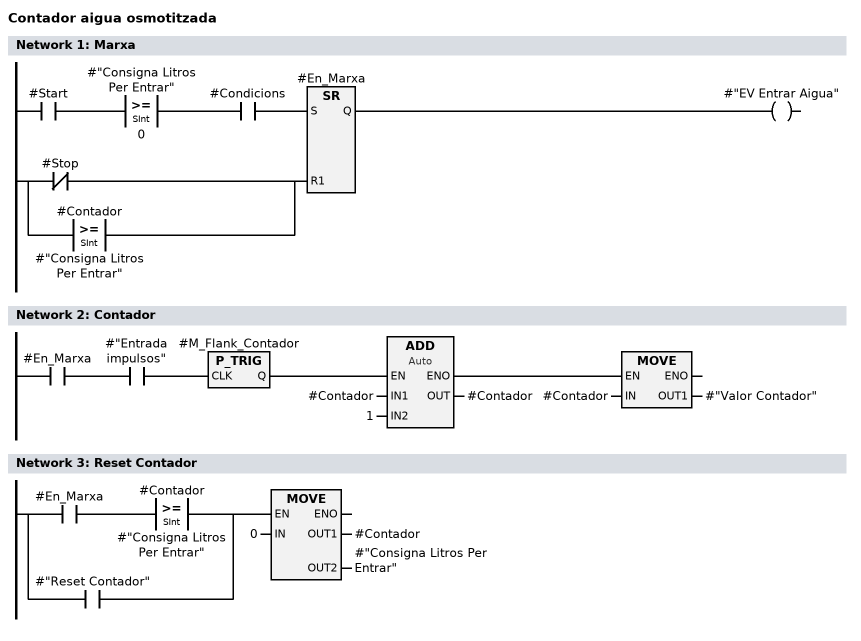
   RUNG wire#powerrail
      Contact( #Start )
      { S7_Templates := "SrcType := SInt" } GE_Contact(in1 := #"Consigna Litros Per Entrar", in2 := 0)
      Contact( #Condicions )
      S_SR(operand := #En_Marxa, r1 := wire#w1)
      Coil( #"EV Entrar Aigua" )
   END_RUNG
   RUNG wire#powerrail
      I_Contact( #Stop )
   END_RUNG wire#w1
   RUNG wire#powerrail
      { S7_Templates := "SrcType := SInt" } GE_Contact(in1 := #Contador, in2 := #"Consigna Litros Per Entrar")
   END_RUNG wire#w1
   // the same network as SCL:
   IF #Start AND (#"Consigna Litros Per Entrar" >= 0) AND #Condicions THEN
       #En_Marxa := TRUE;   // SR flip-flop
   END_IF;
   IF NOT #Stop OR (#Contador >= #"Consigna Litros Per Entrar") THEN #En_Marxa := FALSE; END_IF;
   #"EV Entrar Aigua" := #En_Marxa;
END_REGION

REGION Network 2: Contador
   RUNG wire#powerrail
      Contact( #En_Marxa )
      Contact( #"Entrada impulsos" )
      P_Trig( #M_Flank_Contador )
      Add(in1 := #Contador, in2 := 1, out => #Contador)
      Move(in := #Contador, out1 => #"Valor Contador")
   END_RUNG
   // the same network as SCL:
   #_w1 := #En_Marxa AND #"Entrada impulsos";
   #_w2 := #_w1 AND NOT #M_Flank_Contador;   // rising edge
   #M_Flank_Contador := #_w1;
   IF #_w2 THEN
       #Contador := #Contador + 1;
       #"Valor Contador" := #Contador;
   END_IF;
END_REGION

REGION Network 3: Reset Contador
   RUNG wire#powerrail
      Contact( #En_Marxa )
      { S7_Templates := "SrcType := SInt" } GE_Contact(in1 := #Contador, in2 := #"Consigna Litros Per Entrar")
      wire#w1
      Move(in := 0, out1 => #Contador, out2 => #"Consigna Litros Per Entrar")
   END_RUNG
   RUNG wire#powerrail
      Contact( #"Reset Contador" )
   END_RUNG wire#w1
   // the same network as SCL:
   IF (#En_Marxa AND (#Contador >= #"Consigna Litros Per Entrar")) OR #"Reset Contador" THEN
       #Contador := 0;
       #"Consigna Litros Per Entrar" := 0;
   END_IF;
END_REGION
END_FUNCTION_BLOCK

FUNCTION "FC Elevador" : Void   // FC1, LAD
{ S7_Optimized_Access := 'TRUE' }
VERSION : 0.1
   VAR_INPUT
      "Boto Pujar" : Bool;
      "Boto Baixar" : Bool;
      "Sensor Adalt" : Bool;
      "Sensor Abaix" : Bool;
      Condicio : Bool;
      Termic : Bool;
   END_VAR
   VAR_OUTPUT
      "OUT: Pujar" : Bool;
      "OUT Baixar" : Bool;
   END_VAR
   VAR_TEMP   // added for the SCL form of the ladder/FBD networks
      _w1 : Bool;
   END_VAR
BEGIN

REGION Network 1: Pujar - Baixar
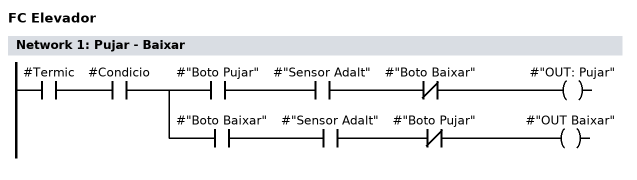
   RUNG wire#powerrail
      Contact( #Termic )
      Contact( #Condicio )
      wire#w1
      Contact( #"Boto Pujar" )
      Contact( #"Sensor Adalt" )
      I_Contact( #"Boto Baixar" )
      Coil( #"OUT: Pujar" )
   END_RUNG
   RUNG wire#w1
      Contact( #"Boto Baixar" )
      Contact( #"Sensor Adalt" )
      I_Contact( #"Boto Pujar" )
      Coil( #"OUT Baixar" )
   END_RUNG
   // the same network as SCL:
   #_w1 := #Termic AND #Condicio;
   #"OUT: Pujar" := #_w1 AND #"Boto Pujar" AND #"Sensor Adalt" AND NOT #"Boto Baixar";
   #"OUT Baixar" := #_w1 AND #"Boto Baixar" AND #"Sensor Adalt" AND NOT #"Boto Pujar";
END_REGION
END_FUNCTION

FUNCTION "Volcar_Desvolcar marmita" : Void   // FC2, LAD
{ S7_Optimized_Access := 'TRUE' }
VERSION : 0.1
   VAR_INPUT
      "Condicio marxa" : Bool;
      "Posicio pales" : Bool;
      "Estat Pales" : Bool;
      "Sensor volcat" : Bool;
      "Sensor desvolcat" : Bool;
      "Boto Volcar" : Bool;
      "Boto Desvolcar" : Bool;
      "Fallo Variador" : Bool;
      "Fallo Termic" : Bool;
   END_VAR
   VAR_IN_OUT
      "OUT: Volcar" : Bool;
      "OUT: Desvolcar" : Bool;
   END_VAR
   VAR_TEMP   // added for the SCL form of the ladder/FBD networks
      _w1 : Bool;
   END_VAR
BEGIN

REGION Network 1: volcar/desvolcar
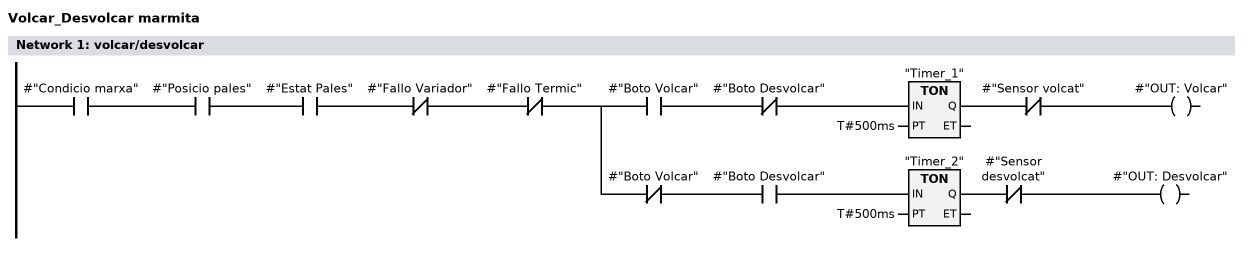
   #_w1 := #"Condicio marxa" AND #"Posicio pales" AND #"Estat Pales" AND NOT #"Fallo Variador" AND NOT #"Fallo Termic";
   "Timer_1".TON(IN := #_w1 AND #"Boto Volcar" AND NOT #"Boto Desvolcar", PT := T#500ms);
   #"OUT: Volcar" := "Timer_1".Q AND NOT #"Sensor volcat";
   "Timer_2".TON(IN := #_w1 AND NOT #"Boto Volcar" AND #"Boto Desvolcar", PT := T#500ms);
   #"OUT: Desvolcar" := "Timer_2".Q AND NOT #"Sensor desvolcat";
END_REGION
END_FUNCTION

FUNCTION "UDINT_TO_TIME" : Void   // FC3, SCL
{ S7_Optimized_Access := 'TRUE' }
VERSION : 0.1
   VAR_INPUT
      Input_1 : UDInt;
   END_VAR
   VAR_OUTPUT
      Output_1 : Time;
   END_VAR
BEGIN
   #Output_1 := T_CONV(#Input_1);
END_FUNCTION

ORGANIZATION_BLOCK "Main"   // OB1, LAD, ProgramCycle
TITLE = "Main Program Sweep (Cycle)"
{ S7_Optimized_Access := 'TRUE' }
VERSION : 0.1
   VAR_INPUT
      Initial_Call : Bool;   // Initial call of this OB
      Remanence : Bool;   // =True, if remanent data are available
   END_VAR
   VAR_TEMP
      Temp_Time : Time;
      Temp_Dint : DInt;
      Status : String;
      "Status Nº Receta" : USInt;
   END_VAR
   VAR_TEMP   // added for the SCL form of the ladder/FBD networks
      _w1 : Bool;
      _w2 : Bool;
   END_VAR
BEGIN

REGION Network 1: Volcar desvolcar marmita
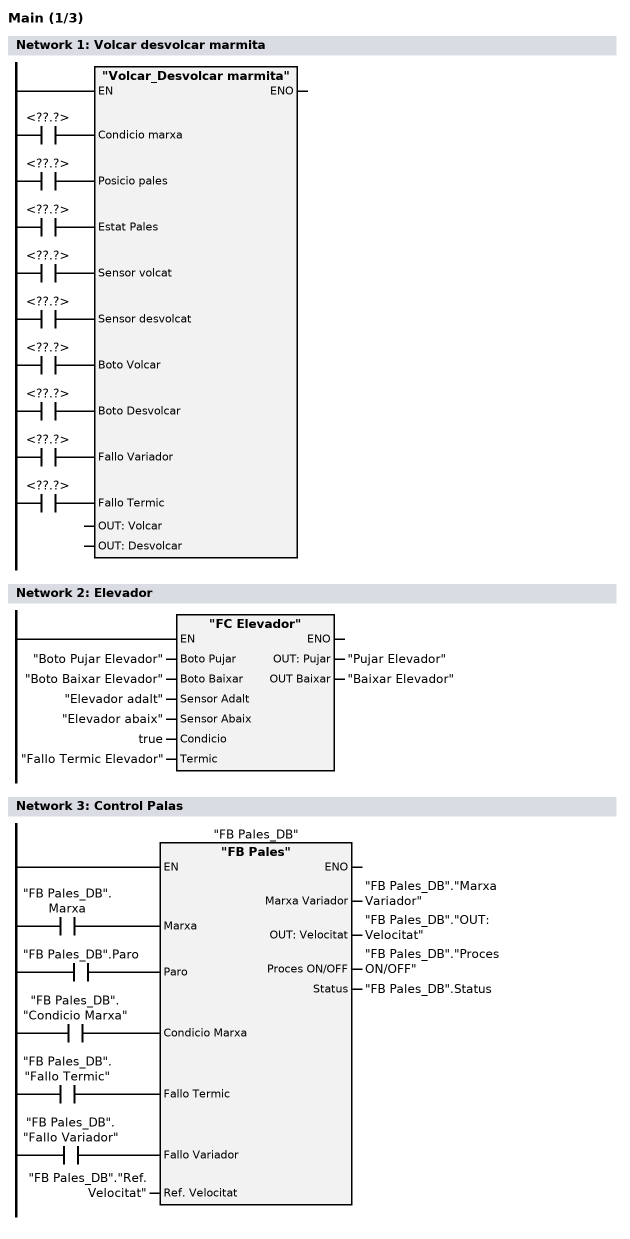
   RUNG wire#powerrail
      "Volcar_Desvolcar marmita"("Condicio marxa" := wire#w1, "Posicio pales" := wire#w2, "Estat Pales" := wire#w3, "Sensor volcat" := wire#w4, "Sensor desvolcat" := wire#w5, "Boto Volcar" := wire#w6, "Boto Desvolcar" := wire#w7, "Fallo Variador" := wire#w8, "Fallo Termic" := wire#w9, "OUT: Volcar" :=, "OUT: Desvolcar" :=)
   END_RUNG
   RUNG wire#powerrail
      Contact(  )
   END_RUNG wire#w1
   RUNG wire#powerrail
      Contact(  )
   END_RUNG wire#w2
   RUNG wire#powerrail
      Contact(  )
   END_RUNG wire#w3
   RUNG wire#powerrail
      Contact(  )
   END_RUNG wire#w4
   RUNG wire#powerrail
      Contact(  )
   END_RUNG wire#w5
   RUNG wire#powerrail
      Contact(  )
   END_RUNG wire#w6
   RUNG wire#powerrail
      Contact(  )
   END_RUNG wire#w7
   RUNG wire#powerrail
      Contact(  )
   END_RUNG wire#w8
   RUNG wire#powerrail
      Contact(  )
   END_RUNG wire#w9
   // the same network as SCL:
   // no checked SCL form for this network; see the picture
END_REGION

REGION Network 2: Elevador
   RUNG wire#powerrail
      "FC Elevador"("Boto Pujar" := "Boto Pujar Elevador", "Boto Baixar" := "Boto Baixar Elevador", "Sensor Adalt" := "Elevador adalt", "Sensor Abaix" := "Elevador abaix", Condicio := true, Termic := "Fallo Termic Elevador", "OUT: Pujar" => "Pujar Elevador", "OUT Baixar" => "Baixar Elevador")
   END_RUNG
   // the same network as SCL:
   "FC Elevador"("Boto Pujar" := "Boto Pujar Elevador",
                 "Boto Baixar" := "Boto Baixar Elevador",
                 "Sensor Adalt" := "Elevador adalt",
                 "Sensor Abaix" := "Elevador abaix",
                 Condicio := true,
                 Termic := "Fallo Termic Elevador",
                 "OUT: Pujar" => "Pujar Elevador",
                 "OUT Baixar" => "Baixar Elevador");
END_REGION

REGION Network 3: Control Palas
   RUNG wire#powerrail
      "FB Pales_DB"(Marxa := wire#w1, Paro := wire#w2, "Condicio Marxa" := wire#w3, "Fallo Termic" := wire#w4, "Fallo Variador" := wire#w5, "Ref. Velocitat" := "FB Pales_DB"."Ref. Velocitat", "Marxa Variador" => "FB Pales_DB"."Marxa Variador", "OUT: Velocitat" => "FB Pales_DB"."OUT: Velocitat", "Proces ON/OFF" => "FB Pales_DB"."Proces ON/OFF", Status => "FB Pales_DB".Status)
   END_RUNG
   RUNG wire#powerrail
      Contact( "FB Pales_DB".Marxa )
   END_RUNG wire#w1
   RUNG wire#powerrail
      Contact( "FB Pales_DB".Paro )
   END_RUNG wire#w2
   RUNG wire#powerrail
      Contact( "FB Pales_DB"."Condicio Marxa" )
   END_RUNG wire#w3
   RUNG wire#powerrail
      Contact( "FB Pales_DB"."Fallo Termic" )
   END_RUNG wire#w4
   RUNG wire#powerrail
      Contact( "FB Pales_DB"."Fallo Variador" )
   END_RUNG wire#w5
   // the same network as SCL:
   "FB Pales_DB"(Marxa := "FB Pales_DB".Marxa,   // "FB Pales"
                 Paro := "FB Pales_DB".Paro,
                 "Condicio Marxa" := "FB Pales_DB"."Condicio Marxa",
                 "Fallo Termic" := "FB Pales_DB"."Fallo Termic",
                 "Fallo Variador" := "FB Pales_DB"."Fallo Variador",
                 "Ref. Velocitat" := "FB Pales_DB"."Ref. Velocitat",
                 "Marxa Variador" => "FB Pales_DB"."Marxa Variador",
                 "OUT: Velocitat" => "FB Pales_DB"."OUT: Velocitat",
                 "Proces ON/OFF" => "FB Pales_DB"."Proces ON/OFF",
                 Status => "FB Pales_DB".Status);
END_REGION

REGION Network 4: Recetas
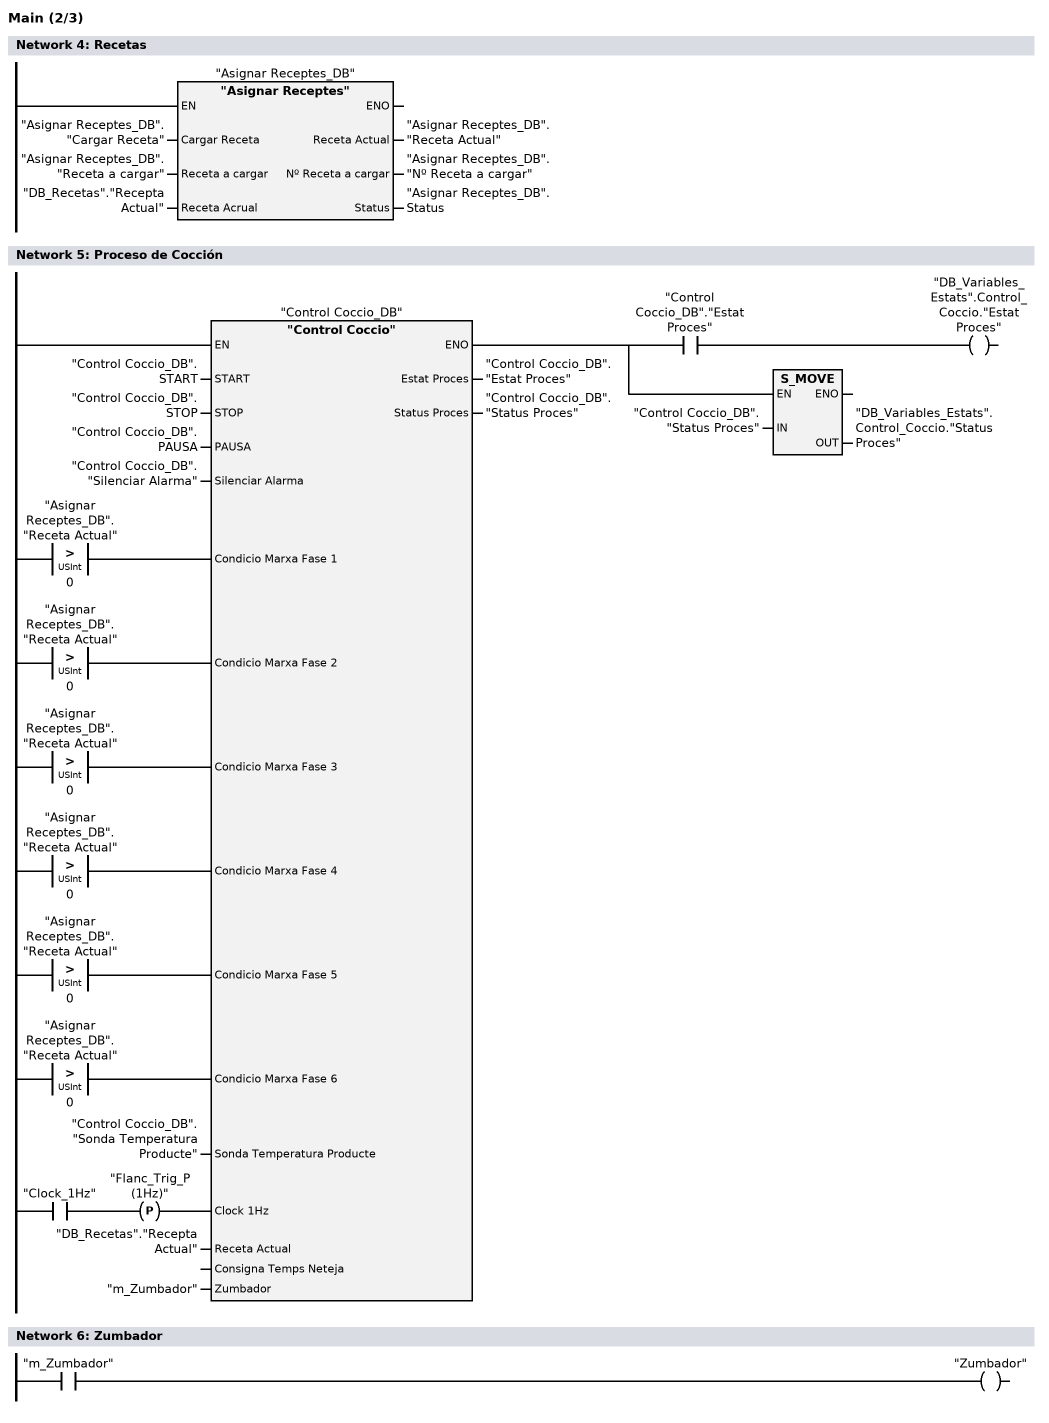
   RUNG wire#powerrail
      "Asignar Receptes_DB"("Cargar Receta" := "Asignar Receptes_DB"."Cargar Receta", "Receta a cargar" := "Asignar Receptes_DB"."Receta a cargar", "Receta Acrual" := "DB_Recetas"."Recepta Actual", "Receta Actual" => "Asignar Receptes_DB"."Receta Actual", "Nº Receta a cargar" => "Asignar Receptes_DB"."Nº Receta a cargar", Status => "Asignar Receptes_DB".Status)
   END_RUNG
   // the same network as SCL:
   "Asignar Receptes_DB"("Cargar Receta" := "Asignar Receptes_DB"."Cargar Receta",   // "Asignar Receptes"
                         "Receta a cargar" := "Asignar Receptes_DB"."Receta a cargar",
                         "Receta Acrual" := "DB_Recetas"."Recepta Actual",
                         "Receta Actual" => "Asignar Receptes_DB"."Receta Actual",
                         "Nº Receta a cargar" => "Asignar Receptes_DB"."Nº Receta a cargar",
                         Status => "Asignar Receptes_DB".Status);
END_REGION

REGION Network 5: Proceso de Cocción
   #_w1 := "Clock_1Hz" AND NOT "Flanc_Trig_P (1Hz)";   // rising edge
   "Flanc_Trig_P (1Hz)" := "Clock_1Hz";
   "Control Coccio_DB"(START := "Control Coccio_DB".START,   // "Control Coccio"
                       STOP := "Control Coccio_DB".STOP,
                       PAUSA := "Control Coccio_DB".PAUSA,
                       "Silenciar Alarma" := "Control Coccio_DB"."Silenciar Alarma",
                       "Condicio Marxa Fase 1" := "Asignar Receptes_DB"."Receta Actual" > 0,
                       "Condicio Marxa Fase 2" := "Asignar Receptes_DB"."Receta Actual" > 0,
                       "Condicio Marxa Fase 3" := "Asignar Receptes_DB"."Receta Actual" > 0,
                       "Condicio Marxa Fase 4" := "Asignar Receptes_DB"."Receta Actual" > 0,
                       "Condicio Marxa Fase 5" := "Asignar Receptes_DB"."Receta Actual" > 0,
                       "Condicio Marxa Fase 6" := "Asignar Receptes_DB"."Receta Actual" > 0,
                       "Sonda Temperatura Producte" := "Control Coccio_DB"."Sonda Temperatura Producte",
                       "Clock 1Hz" := #_w1,
                       "Receta Actual" := "DB_Recetas"."Recepta Actual",
                       Zumbador := "m_Zumbador",
                       "Estat Proces" => "Control Coccio_DB"."Estat Proces",
                       "Status Proces" => "Control Coccio_DB"."Status Proces",
                       ENO => #_w2);
   "DB_Variables_Estats".Control_Coccio."Estat Proces" := #_w2 AND "Control Coccio_DB"."Estat Proces";
   IF #_w2 THEN
       S_MOVE(in := "Control Coccio_DB"."Status Proces",
              out => "DB_Variables_Estats".Control_Coccio."Status Proces");
   END_IF;
END_REGION

REGION Network 6: Zumbador
   RUNG wire#powerrail
      Contact( "m_Zumbador" )
      Coil( "Zumbador" )
   END_RUNG
   // the same network as SCL:
   "Zumbador" := "m_Zumbador";
END_REGION

REGION Network 7: Agua osmotitzada
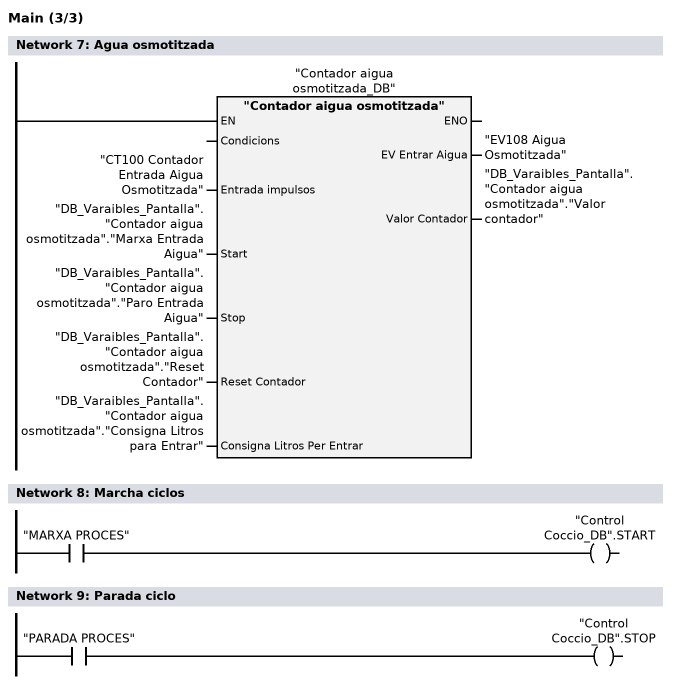
   RUNG wire#powerrail
      "Contador aigua osmotitzada_DB"(Condicions :=, "Entrada impulsos" := "CT100 Contador Entrada Aigua Osmotitzada", Start := "DB_Varaibles_Pantalla"."Contador aigua osmotitzada"."Marxa Entrada Aigua", Stop := "DB_Varaibles_Pantalla"."Contador aigua osmotitzada"."Paro Entrada Aigua", "Reset Contador" := "DB_Varaibles_Pantalla"."Contador aigua osmotitzada"."Reset Contador", "Consigna Litros Per Entrar" := "DB_Varaibles_Pantalla"."Contador aigua osmotitzada"."Consigna Litros para Entrar", "EV Entrar Aigua" => "EV108 Aigua Osmotitzada", "Valor Contador" => "DB_Varaibles_Pantalla"."Contador aigua osmotitzada"."Valor contador")
   END_RUNG
   // the same network as SCL:
   "Contador aigua osmotitzada_DB"("Entrada impulsos" := "CT100 Contador Entrada Aigua Osmotitzada",   // "Contador aigua osmotitzada"
                           Start := "DB_Varaibles_Pantalla"."Contador aigua osmotitzada"."Marxa Entrada Aigua",
                           Stop := "DB_Varaibles_Pantalla"."Contador aigua osmotitzada"."Paro Entrada Aigua",
                           "Reset Contador" := "DB_Varaibles_Pantalla"."Contador aigua osmotitzada"."Reset Contador",
                           "Consigna Litros Per Entrar" := "DB_Varaibles_Pantalla"."Contador aigua osmotitzada"."Consigna Litros para Entrar",
                           "EV Entrar Aigua" => "EV108 Aigua Osmotitzada",
                           "Valor Contador" => "DB_Varaibles_Pantalla"."Contador aigua osmotitzada"."Valor contador");
END_REGION

REGION Network 8: Marcha ciclos
   RUNG wire#powerrail
      Contact( "MARXA PROCES" )
      Coil( "Control Coccio_DB".START )
   END_RUNG
   // the same network as SCL:
   "Control Coccio_DB".START := "MARXA PROCES";
END_REGION

REGION Network 9: Parada ciclo
   RUNG wire#powerrail
      Contact( "PARADA PROCES" )
      Coil( "Control Coccio_DB".STOP )
   END_RUNG
   // the same network as SCL:
   "Control Coccio_DB".STOP := "PARADA PROCES";
END_REGION
END_ORGANIZATION_BLOCK

ORGANIZATION_BLOCK "Cyclic interrupt"   // OB30, LAD, CyclicInterrupt
{ S7_Optimized_Access := 'TRUE' }
VERSION : 0.1
   VAR_INPUT
      Initial_Call : Bool;   // Initial call of this OB
      Event_Count : Int;   // Events discarded
   END_VAR
   VAR_TEMP
      Scaledinput : Real;
      Output : Real;
      State : Int;
      ErrorBits : DWord;
   END_VAR
BEGIN

REGION Network 1
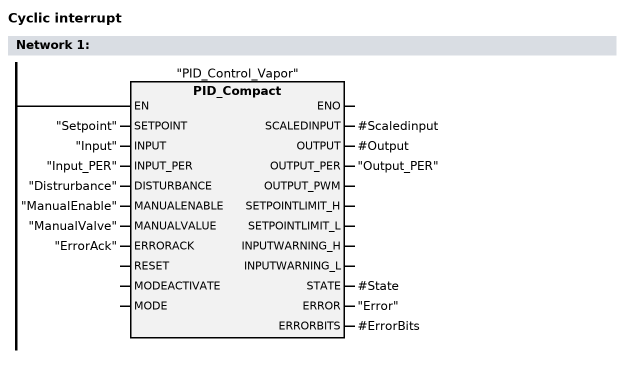
   "PID_Control_Vapor"(Setpoint := "Setpoint",   // PID_Compact
                       Input := "Input",
                       Input_PER := "Input_PER",
                       Disturbance := "Distrurbance",
                       ManualEnable := "ManualEnable",
                       ManualValue := "ManualValve",
                       ErrorAck := "ErrorAck",
                       ScaledInput => #Scaledinput,
                       Output => #Output,
                       Output_PER => "Output_PER",
                       State => #State,
                       Error => "Error",
                       ErrorBits => #ErrorBits);
END_REGION
END_ORGANIZATION_BLOCK